LIN {X 0,Y 302.107,Z 503.378,A -85,B 0,C 180,E1 -16252.782,E2 -16252.782} C_VEL
LIN {X 0,Y 301.296,Z 506.672,A -85,B 0,C 180,E1 -16255.913,E2 -16255.913} C_VEL
LIN {X 0,Y 301.67,Z 508.867,A -85,B 0,C 180,E1 -16256.346,E2 -16256.346} C_VEL
LIN {X 0,Y 303.743,Z 513.97,A -85,B 0,C 180,E1 -16257.676,E2 -16257.676} C_VEL
LIN {X 0,Y 305.482,Z 519.047,A -85,B 0,C 180,E1 -16258.793,E2 -16258.793} C_VEL
LIN {X 0,Y 308.802,Z 531.713,A -85,B 0,C 180,E1 -16261.229,E2 -16261.229} C_VEL
LIN {X 0,Y 310.479,Z 540.82,A -85,B 0,C 180,E1 -16262.787,E2 -16262.787} C_VEL
LIN {X 0,Y 311.403,Z 551.592,A -85,B 0,C 180,E1 -16264.523,E2 -16264.523} C_VEL
LIN {X 0,Y 311.098,Z 562.085,A -85,B 0,C 180,E1 -16266.183,E2 -16266.183} C_VEL
LIN {X 0,Y 309.471,Z 571.424,A -85,B 0,C 180,E1 -16267.642,E2 -16267.642} C_VEL
LIN {X 0,Y 306.369,Z 582.24,A -85,B 0,C 180,E1 -16269.523,E2 -16269.523} C_VEL
LIN {X 0,Y 304.149,Z 589.898,A -85,B 0,C 180,E1 -16271.125,E2 -16271.125} C_VEL
LIN {X 0,Y 301.756,Z 598.006,A -85,B 0,C 180,E1 -16273.167,E2 -16273.167} C_VEL
LIN {X 0,Y 299.626,Z 606.028,A -85,B 0,C 180,E1 -16275.742,E2 -16275.742} C_VEL
LIN {X 0,Y 298.242,Z 611.012,A -85,B 0,C 180,E1 -16277.755,E2 -16277.755} C_VEL
LIN {X 0,Y 297.426,Z 614.951,A -85,B 0,C 180,E1 -16279.792,E2 -16279.792} C_VEL
LIN {X 0,Y 296.891,Z 617.952,A -85,B 0,C 180,E1 -16281.834,E2 -16281.834} C_VEL
LIN {X 0,Y 296.6,Z 620.554,A -85,B 0,C 180,E1 -16284.561,E2 -16284.561} C_VEL
LIN {X 0,Y 296.644,Z 621.226,A -85,B 0,C 180,E1 -16285.924,E2 -16285.924} C_VEL
LIN {X 0,Y 296.862,Z 621.354,A -85,B 0,C 180,E1 -16288.643,E2 -16288.643} C_VEL
LIN {X 0,Y 296.994,Z 620.811,A -85,B 0,C 180,E1 -16290,E2 -16290} C_VEL
LIN {X 0,Y 296.996,Z 619.807,A -85,B 0,C 180,E1 -16291.356,E2 -16291.356} C_VEL
LIN {X 0,Y 296.811,Z 618.326,A -85,B 0,C 180,E1 -16292.714,E2 -16292.714} C_VEL
LIN {X 0,Y 296.889,Z 615.286,A -85,B 0,C 180,E1 -16294.752,E2 -16294.752} C_VEL
LIN {X 0,Y 296.979,Z 611.114,A -85,B 0,C 180,E1 -16296.795,E2 -16296.795} C_VEL
LIN {X 0,Y 297.198,Z 604.706,A -85,B 0,C 180,E1 -16299.185,E2 -16299.185} C_VEL
LIN {X 0,Y 297.65,Z 597.649,A -85,B 0,C 180,E1 -16301.233,E2 -16301.233} C_VEL
LIN {X 0,Y 298.482,Z 588.932,A -85,B 0,C 180,E1 -16303.272,E2 -16303.272} C_VEL
LIN {X 0,Y 299.3,Z 580.046,A -85,B 0,C 180,E1 -16304.969,E2 -16304.969} C_VEL
LIN {X 0,Y 300.483,Z 569.203,A -85,B 0,C 180,E1 -16306.649,E2 -16306.649} C_VEL
LIN {X 0,Y 301.456,Z 558.568,A -85,B 0,C 180,E1 -16307.993,E2 -16307.993} C_VEL
LIN {X 0,Y 300.374,Z 546.843,A -85,B 0,C 180,E1 -16309.237,E2 -16309.237} C_VEL
LIN {X 0,Y 299.033,Z 533.574,A -85,B 0,C 180,E1 -16310.352,E2 -16310.352} C_VEL
LIN {X 0,Y 297.686,Z 520.117,A -85,B 0,C 180,E1 -16311.216,E2 -16311.216} C_VEL
LIN {X 0,Y 297.486,Z 517.081,A -85,B 0,C 180,E1 -16311.389,E2 -16311.389} C_VEL
LIN {X 0,Y 298.225,Z 509.911,A -85,B 0,C 180,E1 -16315.793,E2 -16315.793} C_VEL
LIN {X 0,Y 299.087,Z 503.762,A -85,B 0,C 180,E1 -16319.607,E2 -16319.607} C_VEL
LIN {X 0,Y 300.024,Z 497.747,A -85,B 0,C 180,E1 -16323.4,E2 -16323.4} C_VEL
LIN {X 0,Y 300.596,Z 494.041,A -85,B 0,C 180,E1 -16325.768,E2 -16325.768} C_VEL
LIN {X 0,Y 300.422,Z 490.212,A -85,B 0,C 180,E1 -16328.311,E2 -16328.311} C_VEL
LIN {X 0,Y 299.452,Z 484.838,A -85,B 0,C 180,E1 -16332.082,E2 -16332.082} C_VEL
LIN {X 0,Y 298.523,Z 479.301,A -85,B 0,C 180,E1 -16336.189,E2 -16336.189} C_VEL
LIN {X 0,Y 298.427,Z 479.312,A -85,B 0,C 180,E1 -16340.517,E2 -16340.517} C_VEL
LIN {X 0,Y 298.432,Z 479.308,A -85,B 0,C 180,E1 -16343.932,E2 -16343.932} C_VEL
LIN {X 0,Y 298.394,Z 479.313,A -85,B 0,C 180,E1 -16347.984,E2 -16347.984} C_VEL
LIN {X 0,Y 298.458,Z 479.304,A -85,B 0,C 180,E1 -16351.904,E2 -16351.904} C_VEL
LIN {X 0,Y 298.484,Z 479.304,A -85,B 0,C 180,E1 -16354.924,E2 -16354.924} C_VEL
LIN {X 0,Y 298.451,Z 479.305,A -85,B 0,C 180,E1 -16359.316,E2 -16359.316} C_VEL
LIN {X 0,Y 298.539,Z 479.296,A -85,B 0,C 180,E1 -16362.18,E2 -16362.18} C_VEL
LIN {X 0,Y 298.595,Z 479.29,A -85,B 0,C 180,E1 -16364.995,E2 -16364.995} C_VEL
LIN {X 0,Y 298.595,Z 479.288,A -85,B 0,C 180,E1 -16369.147,E2 -16369.147} C_VEL
LIN {X 0,Y 298.76,Z 479.268,A -85,B 0,C 180,E1 -16371.886,E2 -16371.886} C_VEL
LIN {X 0,Y 298.661,Z 479.284,A -85,B 0,C 180,E1 -16374.599,E2 -16374.599} C_VEL
LIN {X 0,Y 298.925,Z 479.25,A -85,B 0,C 180,E1 -16378.653,E2 -16378.653} C_VEL
LIN {X 0,Y 298.926,Z 479.247,A -85,B 0,C 180,E1 -16381.347,E2 -16381.347} C_VEL
LIN {X 0,Y 298.8,Z 479.264,A -85,B 0,C 180,E1 -16386.754,E2 -16386.754} C_VEL
LIN {X 0,Y 298.682,Z 479.277,A -85,B 0,C 180,E1 -16389.481,E2 -16389.481} C_VEL
LIN {X 0,Y 298.554,Z 479.293,A -85,B 0,C 180,E1 -16393.616,E2 -16393.616} C_VEL
LIN {X 0,Y 298.55,Z 479.298,A -85,B 0,C 180,E1 -16396.409,E2 -16396.409} C_VEL
LIN {X 0,Y 298.514,Z 479.298,A -85,B 0,C 180,E1 -16399.655,E2 -16399.655} C_VEL
LIN {X 0,Y 298.459,Z 479.304,A -85,B 0,C 180,E1 -16403.598,E2 -16403.598} C_VEL
LIN {X 0,Y 298.491,Z 479.304,A -85,B 0,C 180,E1 -16406.575,E2 -16406.575} C_VEL
LIN {X 0,Y 298.423,Z 479.31,A -85,B 0,C 180,E1 -16409.641,E2 -16409.641} C_VEL
LIN {X 0,Y 298.398,Z 479.313,A -85,B 0,C 180,E1 -16412.8,E2 -16412.8} C_VEL
LIN {X 0,Y 298.448,Z 479.307,A -85,B 0,C 180,E1 -16416.808,E2 -16416.808} C_VEL
LIN {X 0,Y 298.411,Z 479.311,A -85,B 0,C 180,E1 -16419.486,E2 -16419.486} C_VEL
LIN {X 0,Y 298.4,Z 479.312,A -85,B 0,C 180,E1 -16423.104,E2 -16423.104} C_VEL
LIN {X 0,Y 298.405,Z 479.312,A -85,B 0,C 180,E1 -16426.921,E2 -16426.921} C_VEL
LIN {X 0,Y 298.418,Z 479.309,A -85,B 0,C 180,E1 -16431.004,E2 -16431.004} C_VEL
LIN {X 0,Y 298.435,Z 479.311,A -85,B 0,C 180,E1 -16433.933,E2 -16433.933} C_VEL
LIN {X 0,Y 298.397,Z 479.316,A -85,B 0,C 180,E1 -16437.984,E2 -16437.984} C_VEL
LIN {X 0,Y 298.462,Z 479.307,A -85,B 0,C 180,E1 -16441.904,E2 -16441.904} C_VEL
LIN {X 0,Y 298.489,Z 479.301,A -85,B 0,C 180,E1 -16444.924,E2 -16444.924} C_VEL
LIN {X 0,Y 298.454,Z 479.305,A -85,B 0,C 180,E1 -16449.316,E2 -16449.316} C_VEL
LIN {X 0,Y 298.542,Z 479.299,A -85,B 0,C 180,E1 -16452.18,E2 -16452.18} C_VEL
LIN {X 0,Y 298.597,Z 479.287,A -85,B 0,C 180,E1 -16454.995,E2 -16454.995} C_VEL
LIN {X 0,Y 298.595,Z 479.288,A -85,B 0,C 180,E1 -16459.147,E2 -16459.147} C_VEL
LIN {X 0,Y 298.717,Z 479.276,A -85,B 0,C 180,E1 -16461.885,E2 -16461.885} C_VEL
LIN {X 0,Y 298.648,Z 479.281,A -85,B 0,C 180,E1 -16464.599,E2 -16464.599} C_VEL
LIN {X 0,Y 298.928,Z 479.247,A -85,B 0,C 180,E1 -16468.653,E2 -16468.653} C_VEL
LIN {X 0,Y 298.926,Z 479.247,A -85,B 0,C 180,E1 -16471.347,E2 -16471.347} C_VEL
LIN {X 0,Y 298.791,Z 479.263,A -85,B 0,C 180,E1 -16476.754,E2 -16476.754} C_VEL
LIN {X 0,Y 298.64,Z 479.284,A -85,B 0,C 180,E1 -16479.482,E2 -16479.482} C_VEL
LIN {X 0,Y 298.556,Z 479.294,A -85,B 0,C 180,E1 -16483.615,E2 -16483.615} C_VEL
LIN {X 0,Y 298.553,Z 479.294,A -85,B 0,C 180,E1 -16486.409,E2 -16486.409} C_VEL
LIN {X 0,Y 298.516,Z 479.301,A -85,B 0,C 180,E1 -16489.655,E2 -16489.655} C_VEL
LIN {X 0,Y 298.461,Z 479.307,A -85,B 0,C 180,E1 -16493.598,E2 -16493.598} C_VEL
LIN {X 0,Y 298.49,Z 479.301,A -85,B 0,C 180,E1 -16496.575,E2 -16496.575} C_VEL
LIN {X 0,Y 298.42,Z 479.313,A -85,B 0,C 180,E1 -16499.641,E2 -16499.641} C_VEL
LIN {X 0,Y 298.399,Z 479.312,A -85,B 0,C 180,E1 -16502.8,E2 -16502.8} C_VEL
LIN {X 0,Y 298.454,Z 479.305,A -85,B 0,C 180,E1 -16506.809,E2 -16506.809} C_VEL
LIN {X 0,Y 298.412,Z 479.313,A -85,B 0,C 180,E1 -16509.486,E2 -16509.486} C_VEL
LIN {X 0,Y 298.402,Z 479.312,A -85,B 0,C 180,E1 -16513.103,E2 -16513.103} C_VEL
LIN {X 0,Y 298.406,Z 479.311,A -85,B 0,C 180,E1 -16516.921,E2 -16516.921} C_VEL
LIN {X 0,Y 298.392,Z 479.313,A -85,B 0,C 180,E1 -16521.01,E2 -16521.01} C_VEL
LIN {X 0,Y 298.304,Z 479.327,A -85,B 0,C 180,E1 -16523.914,E2 -16523.914} C_VEL
LIN {X 0,Y 297.986,Z 479.364,A -85,B 0,C 180,E1 -16527.149,E2 -16527.149} C_VEL
LIN {X 0,Y 297.642,Z 479.407,A -85,B 0,C 180,E1 -16530.887,E2 -16530.887} C_VEL
LIN {X 0,Y 297.319,Z 479.451,A -85,B 0,C 180,E1 -16533.928,E2 -16533.928} C_VEL
LIN {X 0,Y 297.221,Z 479.745,A -85,B 0,C 180,E1 -16534.81,E2 -16534.81} C_VEL
LIN {X 0,Y 297.105,Z 483.567,A -85,B 0,C 180,E1 -16538.89,E2 -16538.89} C_VEL
LIN {X 0,Y 299.629,Z 496.768,A -85,B 0,C 180,E1 -16539.757,E2 -16539.757} C_VEL
LIN {X 0,Y 302.182,Z 509.983,A -85,B 0,C 180,E1 -16540.89,E2 -16540.89} C_VEL
LIN {X 0,Y 302.831,Z 515.047,A -85,B 0,C 180,E1 -16541.391,E2 -16541.391} C_VEL
LIN {X 0,Y 301.789,Z 527.176,A -85,B 0,C 180,E1 -16542.709,E2 -16542.709} C_VEL
LIN {X 0,Y 300.718,Z 538.429,A -85,B 0,C 180,E1 -16544.235,E2 -16544.235} C_VEL
LIN {X 0,Y 299.799,Z 547.646,A -85,B 0,C 180,E1 -16545.75,E2 -16545.75} C_VEL
LIN {X 0,Y 298.768,Z 557.725,A -85,B 0,C 180,E1 -16547.777,E2 -16547.777} C_VEL
LIN {X 0,Y 298,Z 565.938,A -85,B 0,C 180,E1 -16549.812,E2 -16549.812} C_VEL
LIN {X 0,Y 297.448,Z 572.604,A -85,B 0,C 180,E1 -16551.85,E2 -16551.85} C_VEL
LIN {X 0,Y 297.056,Z 578.093,A -85,B 0,C 180,E1 -16553.957,E2 -16553.957} C_VEL
LIN {X 0,Y 296.938,Z 582.134,A -85,B 0,C 180,E1 -16555.928,E2 -16555.928} C_VEL
LIN {X 0,Y 296.865,Z 583.076,A -85,B 0,C 180,E1 -16556.475,E2 -16556.475} C_VEL
LIN {X 0,Y 296.11,Z 584.795,A -85,B 0,C 180,E1 -16557.557,E2 -16557.557} C_VEL
LIN {X 0,Y 293.211,Z 587.005,A -85,B 0,C 180,E1 -16559.351,E2 -16559.351} C_VEL
LIN {X 0,Y 290.88,Z 588.266,A -85,B 0,C 180,E1 -16560.828,E2 -16560.828} C_VEL
LIN {X 0,Y 289.989,Z 588.981,A -85,B 0,C 180,E1 -16561.979,E2 -16561.979} C_VEL
LIN {X 0,Y 289.972,Z 589.117,A -85,B 0,C 180,E1 -16562.369,E2 -16562.369} C_VEL
LIN {X 0,Y 290.338,Z 589.507,A -85,B 0,C 180,E1 -16564.164,E2 -16564.164} C_VEL
LIN {X 0,Y 290.839,Z 588.823,A -85,B 0,C 180,E1 -16566.939,E2 -16566.939} C_VEL
LIN {X 0,Y 292.244,Z 586.468,A -85,B 0,C 180,E1 -16569.691,E2 -16569.691} C_VEL
LIN {X 0,Y 293.876,Z 582.596,A -85,B 0,C 180,E1 -16572.429,E2 -16572.429} C_VEL
LIN {X 0,Y 295.649,Z 578.513,A -85,B 0,C 180,E1 -16574.454,E2 -16574.454} C_VEL
LIN {X 0,Y 297.634,Z 573.361,A -85,B 0,C 180,E1 -16576.46,E2 -16576.46} C_VEL
LIN {X 0,Y 300.395,Z 565.915,A -85,B 0,C 180,E1 -16578.765,E2 -16578.765} C_VEL
LIN {X 0,Y 303.37,Z 557.96,A -85,B 0,C 180,E1 -16580.688,E2 -16580.688} C_VEL
LIN {X 0,Y 306.517,Z 548.367,A -85,B 0,C 180,E1 -16582.585,E2 -16582.585} C_VEL
LIN {X 0,Y 309.442,Z 538.773,A -85,B 0,C 180,E1 -16584.13,E2 -16584.13} C_VEL
LIN {X 0,Y 310.422,Z 534.633,A -85,B 0,C 180,E1 -16584.744,E2 -16584.744} C_VEL
LIN {X 0,Y 308.526,Z 525.506,A -85,B 0,C 180,E1 -16586.831,E2 -16586.831} C_VEL
LIN {X 0,Y 306.405,Z 519.377,A -85,B 0,C 180,E1 -16588.413,E2 -16588.413} C_VEL
LIN {X 0,Y 303.715,Z 513.027,A -85,B 0,C 180,E1 -16590.241,E2 -16590.241} C_VEL
LIN {X 0,Y 302.235,Z 509.907,A -85,B 0,C 180,E1 -16591.215,E2 -16591.215} C_VEL
LIN {X 0,Y 300.186,Z 506.257,A -85,B 0,C 180,E1 -16592.58,E2 -16592.58} C_VEL
LIN {X 0,Y 298.449,Z 503.948,A -85,B 0,C 180,E1 -16593.694,E2 -16593.694} C_VEL
LIN {X 0,Y 297.462,Z 501.682,A -85,B 0,C 180,E1 -16594.544,E2 -16594.544} C_VEL
LIN {X 0,Y 295.377,Z 499.782,A -85,B 0,C 180,E1 -16596.004,E2 -16596.004} C_VEL
LIN {X 0,Y 294.153,Z 496.998,A -85,B 0,C 180,E1 -16597.437,E2 -16597.437} C_VEL
LIN {X 0,Y 294.39,Z 497.575,A -85,B 0,C 180,E1 -16600.187,E2 -16600.187} C_VEL
LIN {X 0,Y 294.661,Z 498.846,A -85,B 0,C 180,E1 -16603.764,E2 -16603.764} C_VEL
LIN {X 0,Y 295.006,Z 500.89,A -85,B 0,C 180,E1 -16607.606,E2 -16607.606} C_VEL
LIN {X 0,Y 295.213,Z 502.538,A -85,B 0,C 180,E1 -16610,E2 -16610} C_VEL
LIN {X 0,Y 295.074,Z 505.124,A -85,B 0,C 180,E1 -16613.035,E2 -16613.035} C_VEL
LIN {X 0,Y 295.688,Z 508.225,A -85,B 0,C 180,E1 -16613.913,E2 -16613.913} C_VEL
LIN {X 0,Y 297.728,Z 512.868,A -85,B 0,C 180,E1 -16615.491,E2 -16615.491} C_VEL
LIN {X 0,Y 298.885,Z 516.803,A -85,B 0,C 180,E1 -16616.493,E2 -16616.493} C_VEL
LIN {X 0,Y 299.627,Z 518.634,A -85,B 0,C 180,E1 -16617.017,E2 -16617.017} C_VEL
LIN {X 0,Y 301.626,Z 526.286,A -85,B 0,C 180,E1 -16618.733,E2 -16618.733} C_VEL
LIN {X 0,Y 303.297,Z 533.136,A -85,B 0,C 180,E1 -16620.169,E2 -16620.169} C_VEL
LIN {X 0,Y 304.843,Z 542.716,A -85,B 0,C 180,E1 -16621.97,E2 -16621.97} C_VEL
LIN {X 0,Y 305.551,Z 553.087,A -85,B 0,C 180,E1 -16623.772,E2 -16623.772} C_VEL
LIN {X 0,Y 305.105,Z 563.405,A -85,B 0,C 180,E1 -16625.504,E2 -16625.504} C_VEL
LIN {X 0,Y 303.053,Z 573.235,A -85,B 0,C 180,E1 -16627.142,E2 -16627.142} C_VEL
LIN {X 0,Y 299.851,Z 583.62,A -85,B 0,C 180,E1 -16629.057,E2 -16629.057} C_VEL
LIN {X 0,Y 297.012,Z 592.414,A -85,B 0,C 180,E1 -16631.057,E2 -16631.057} C_VEL
LIN {X 0,Y 294.771,Z 599.512,A -85,B 0,C 180,E1 -16633.018,E2 -16633.018} C_VEL
LIN {X 0,Y 292.767,Z 606.445,A -85,B 0,C 180,E1 -16635.4,E2 -16635.4} C_VEL
LIN {X 0,Y 291.287,Z 611.213,A -85,B 0,C 180,E1 -16637.458,E2 -16637.458} C_VEL
LIN {X 0,Y 290.195,Z 616.022,A -85,B 0,C 180,E1 -16640.239,E2 -16640.239} C_VEL
LIN {X 0,Y 289.605,Z 619.229,A -85,B 0,C 180,E1 -16643.031,E2 -16643.031} C_VEL
LIN {X 0,Y 289.536,Z 620.209,A -85,B 0,C 180,E1 -16644.428,E2 -16644.428} C_VEL
LIN {X 0,Y 289.555,Z 620.796,A -85,B 0,C 180,E1 -16645.824,E2 -16645.824} C_VEL
LIN {X 0,Y 289.773,Z 620.785,A -85,B 0,C 180,E1 -16648.61,E2 -16648.61} C_VEL
LIN {X 0,Y 289.94,Z 620.14,A -85,B 0,C 180,E1 -16650,E2 -16650} C_VEL
LIN {X 0,Y 289.938,Z 619.046,A -85,B 0,C 180,E1 -16651.389,E2 -16651.389} C_VEL
LIN {X 0,Y 289.741,Z 617.499,A -85,B 0,C 180,E1 -16652.78,E2 -16652.78} C_VEL
LIN {X 0,Y 289.839,Z 614.321,A -85,B 0,C 180,E1 -16654.868,E2 -16654.868} C_VEL
LIN {X 0,Y 289.926,Z 610.008,A -85,B 0,C 180,E1 -16656.961,E2 -16656.961} C_VEL
LIN {X 0,Y 290.174,Z 603.387,A -85,B 0,C 180,E1 -16659.409,E2 -16659.409} C_VEL
LIN {X 0,Y 290.668,Z 596.139,A -85,B 0,C 180,E1 -16661.506,E2 -16661.506} C_VEL
LIN {X 0,Y 291.538,Z 587.211,A -85,B 0,C 180,E1 -16663.594,E2 -16663.594} C_VEL
LIN {X 0,Y 292.568,Z 576.541,A -85,B 0,C 180,E1 -16665.583,E2 -16665.583} C_VEL
LIN {X 0,Y 293.789,Z 565.673,A -85,B 0,C 180,E1 -16667.219,E2 -16667.219} C_VEL
LIN {X 0,Y 294.292,Z 557.319,A -85,B 0,C 180,E1 -16668.266,E2 -16668.266} C_VEL
LIN {X 0,Y 293.043,Z 544.534,A -85,B 0,C 180,E1 -16669.619,E2 -16669.619} C_VEL
LIN {X 0,Y 291.658,Z 530.634,A -85,B 0,C 180,E1 -16670.777,E2 -16670.777} C_VEL
LIN {X 0,Y 290.419,Z 516.721,A -85,B 0,C 180,E1 -16671.656,E2 -16671.656} C_VEL
LIN {X 0,Y 291.116,Z 510.248,A -85,B 0,C 180,E1 -16675.756,E2 -16675.756} C_VEL
LIN {X 0,Y 292.082,Z 503.639,A -85,B 0,C 180,E1 -16679.977,E2 -16679.977} C_VEL
LIN {X 0,Y 293.164,Z 496.988,A -85,B 0,C 180,E1 -16684.289,E2 -16684.289} C_VEL
LIN {X 0,Y 293.549,Z 493.273,A -85,B 0,C 180,E1 -16686.765,E2 -16686.765} C_VEL
LIN {X 0,Y 292.981,Z 488.85,A -85,B 0,C 180,E1 -16689.86,E2 -16689.86} C_VEL
LIN {X 0,Y 292.002,Z 483.47,A -85,B 0,C 180,E1 -16693.776,E2 -16693.776} C_VEL
LIN {X 0,Y 291.486,Z 480.178,A -85,B 0,C 180,E1 -16696.33,E2 -16696.33} C_VEL
LIN {X 0,Y 291.403,Z 480.187,A -85,B 0,C 180,E1 -16700.513,E2 -16700.513} C_VEL
LIN {X 0,Y 291.428,Z 480.183,A -85,B 0,C 180,E1 -16702.923,E2 -16702.923} C_VEL
LIN {X 0,Y 291.345,Z 480.193,A -85,B 0,C 180,E1 -16706.302,E2 -16706.302} C_VEL
LIN {X 0,Y 291.384,Z 480.188,A -85,B 0,C 180,E1 -16710.261,E2 -16710.261} C_VEL
LIN {X 0,Y 291.413,Z 480.184,A -85,B 0,C 180,E1 -16714.272,E2 -16714.272} C_VEL
LIN {X 0,Y 291.383,Z 480.187,A -85,B 0,C 180,E1 -16717.3,E2 -16717.3} C_VEL
LIN {X 0,Y 291.459,Z 480.178,A -85,B 0,C 180,E1 -16720.27,E2 -16720.27} C_VEL
LIN {X 0,Y 291.556,Z 480.17,A -85,B 0,C 180,E1 -16724.624,E2 -16724.624} C_VEL
LIN {X 0,Y 291.538,Z 480.168,A -85,B 0,C 180,E1 -16728.881,E2 -16728.881} C_VEL
LIN {X 0,Y 291.71,Z 480.145,A -85,B 0,C 180,E1 -16731.689,E2 -16731.689} C_VEL
LIN {X 0,Y 291.632,Z 480.16,A -85,B 0,C 180,E1 -16734.469,E2 -16734.469} C_VEL
LIN {X 0,Y 291.891,Z 480.127,A -85,B 0,C 180,E1 -16738.621,E2 -16738.621} C_VEL
LIN {X 0,Y 291.892,Z 480.123,A -85,B 0,C 180,E1 -16741.38,E2 -16741.38} C_VEL
LIN {X 0,Y 291.748,Z 480.142,A -85,B 0,C 180,E1 -16746.918,E2 -16746.918} C_VEL
LIN {X 0,Y 291.631,Z 480.156,A -85,B 0,C 180,E1 -16749.712,E2 -16749.712} C_VEL
LIN {X 0,Y 291.524,Z 480.17,A -85,B 0,C 180,E1 -16753.951,E2 -16753.951} C_VEL
LIN {X 0,Y 291.489,Z 480.175,A -85,B 0,C 180,E1 -16756.818,E2 -16756.818} C_VEL
LIN {X 0,Y 291.452,Z 480.179,A -85,B 0,C 180,E1 -16759.875,E2 -16759.875} C_VEL
LIN {X 0,Y 291.402,Z 480.187,A -85,B 0,C 180,E1 -16764.205,E2 -16764.205} C_VEL
LIN {X 0,Y 291.424,Z 480.181,A -85,B 0,C 180,E1 -16767.272,E2 -16767.272} C_VEL
LIN {X 0,Y 291.339,Z 480.195,A -85,B 0,C 180,E1 -16770.437,E2 -16770.437} C_VEL
LIN {X 0,Y 291.347,Z 480.19,A -85,B 0,C 180,E1 -16773.699,E2 -16773.699} C_VEL
LIN {X 0,Y 291.383,Z 480.186,A -85,B 0,C 180,E1 -16777.256,E2 -16777.256} C_VEL
LIN {X 0,Y 291.336,Z 480.193,A -85,B 0,C 180,E1 -16780.643,E2 -16780.643} C_VEL
LIN {X 0,Y 291.292,Z 480.201,A -85,B 0,C 180,E1 -16784.402,E2 -16784.402} C_VEL
LIN {X 0,Y 291.329,Z 480.196,A -85,B 0,C 180,E1 -16788.405,E2 -16788.405} C_VEL
LIN {X 0,Y 291.367,Z 480.187,A -85,B 0,C 180,E1 -16791.161,E2 -16791.161} C_VEL
LIN {X 0,Y 291.388,Z 480.187,A -85,B 0,C 180,E1 -16794.63,E2 -16794.63} C_VEL
LIN {X 0,Y 291.374,Z 480.19,A -85,B 0,C 180,E1 -16797.951,E2 -16797.951} C_VEL
LIN {X 0,Y 291.38,Z 480.186,A -85,B 0,C 180,E1 -16801.158,E2 -16801.158} C_VEL
LIN {X 0,Y 291.418,Z 480.186,A -85,B 0,C 180,E1 -16804.272,E2 -16804.272} C_VEL
LIN {X 0,Y 291.385,Z 480.185,A -85,B 0,C 180,E1 -16807.3,E2 -16807.3} C_VEL
LIN {X 0,Y 291.462,Z 480.18,A -85,B 0,C 180,E1 -16810.271,E2 -16810.271} C_VEL
LIN {X 0,Y 291.559,Z 480.165,A -85,B 0,C 180,E1 -16814.624,E2 -16814.624} C_VEL
LIN {X 0,Y 291.539,Z 480.167,A -85,B 0,C 180,E1 -16818.881,E2 -16818.881} C_VEL
LIN {X 0,Y 291.668,Z 480.153,A -85,B 0,C 180,E1 -16821.687,E2 -16821.687} C_VEL
LIN {X 0,Y 291.617,Z 480.158,A -85,B 0,C 180,E1 -16824.468,E2 -16824.468} C_VEL
LIN {X 0,Y 291.894,Z 480.123,A -85,B 0,C 180,E1 -16828.62,E2 -16828.62} C_VEL
LIN {X 0,Y 291.893,Z 480.123,A -85,B 0,C 180,E1 -16831.38,E2 -16831.38} C_VEL
LIN {X 0,Y 291.739,Z 480.142,A -85,B 0,C 180,E1 -16836.918,E2 -16836.918} C_VEL
LIN {X 0,Y 291.579,Z 480.165,A -85,B 0,C 180,E1 -16839.714,E2 -16839.714} C_VEL
LIN {X 0,Y 291.526,Z 480.173,A -85,B 0,C 180,E1 -16843.95,E2 -16843.95} C_VEL
LIN {X 0,Y 291.491,Z 480.173,A -85,B 0,C 180,E1 -16846.818,E2 -16846.818} C_VEL
LIN {X 0,Y 291.454,Z 480.182,A -85,B 0,C 180,E1 -16849.875,E2 -16849.875} C_VEL
LIN {X 0,Y 291.404,Z 480.186,A -85,B 0,C 180,E1 -16854.205,E2 -16854.205} C_VEL
LIN {X 0,Y 291.423,Z 480.182,A -85,B 0,C 180,E1 -16857.272,E2 -16857.272} C_VEL
LIN {X 0,Y 291.338,Z 480.191,A -85,B 0,C 180,E1 -16860.437,E2 -16860.437} C_VEL
LIN {X 0,Y 291.348,Z 480.194,A -85,B 0,C 180,E1 -16863.698,E2 -16863.698} C_VEL
LIN {X 0,Y 291.388,Z 480.187,A -85,B 0,C 180,E1 -16867.256,E2 -16867.256} C_VEL
LIN {X 0,Y 291.337,Z 480.191,A -85,B 0,C 180,E1 -16870.642,E2 -16870.642} C_VEL
LIN {X 0,Y 291.293,Z 480.198,A -85,B 0,C 180,E1 -16874.402,E2 -16874.402} C_VEL
LIN {X 0,Y 291.329,Z 480.192,A -85,B 0,C 180,E1 -16878.404,E2 -16878.404} C_VEL
LIN {X 0,Y 291.338,Z 480.193,A -85,B 0,C 180,E1 -16881.155,E2 -16881.155} C_VEL
LIN {X 0,Y 291.33,Z 480.193,A -85,B 0,C 180,E1 -16882.907,E2 -16882.907} C_VEL
LIN {X 0,Y 291.028,Z 480.23,A -85,B 0,C 180,E1 -16886.26,E2 -16886.26} C_VEL
LIN {X 0,Y 290.709,Z 480.273,A -85,B 0,C 180,E1 -16889.49,E2 -16889.49} C_VEL
LIN {X 0,Y 290.366,Z 480.319,A -85,B 0,C 180,E1 -16892.621,E2 -16892.621} C_VEL
LIN {X 0,Y 290.238,Z 480.333,A -85,B 0,C 180,E1 -16894.159,E2 -16894.159} C_VEL
LIN {X 0,Y 290.085,Z 481.171,A -85,B 0,C 180,E1 -16895.678,E2 -16895.678} C_VEL
LIN {X 0,Y 290.038,Z 483.915,A -85,B 0,C 180,E1 -16898.64,E2 -16898.64} C_VEL
LIN {X 0,Y 292.535,Z 497.318,A -85,B 0,C 180,E1 -16899.547,E2 -16899.547} C_VEL
LIN {X 0,Y 295.269,Z 511.479,A -85,B 0,C 180,E1 -16900.806,E2 -16900.806} C_VEL
LIN {X 0,Y 295.769,Z 516.21,A -85,B 0,C 180,E1 -16901.289,E2 -16901.289} C_VEL
LIN {X 0,Y 294.616,Z 528.976,A -85,B 0,C 180,E1 -16902.748,E2 -16902.748} C_VEL
LIN {X 0,Y 293.562,Z 539.263,A -85,B 0,C 180,E1 -16904.197,E2 -16904.197} C_VEL
LIN {X 0,Y 292.662,Z 548.424,A -85,B 0,C 180,E1 -16905.75,E2 -16905.75} C_VEL
LIN {X 0,Y 291.654,Z 558.437,A -85,B 0,C 180,E1 -16907.828,E2 -16907.828} C_VEL
LIN {X 0,Y 290.874,Z 566.617,A -85,B 0,C 180,E1 -16909.911,E2 -16909.911} C_VEL
LIN {X 0,Y 290.393,Z 572.217,A -85,B 0,C 180,E1 -16911.65,E2 -16911.65} C_VEL
LIN {X 0,Y 289.95,Z 578.397,A -85,B 0,C 180,E1 -16914.03,E2 -16914.03} C_VEL
LIN {X 0,Y 289.789,Z 583.133,A -85,B 0,C 180,E1 -16916.452,E2 -16916.452} C_VEL
LIN {X 0,Y 289.673,Z 586.207,A -85,B 0,C 180,E1 -16918.61,E2 -16918.61} C_VEL
LIN {X 0,Y 289.71,Z 587.658,A -85,B 0,C 180,E1 -16920,E2 -16920} C_VEL
LIN {X 0,Y 289.972,Z 589.117,A -85,B 0,C 180,E1 -16922.369,E2 -16922.369} C_VEL
LIN {X 0,Y 289.5,Z 589.557,A -85,B 0,C 180,E1 -16923.53,E2 -16923.53} C_VEL
LIN {X 0,Y 286.985,Z 589.879,A -85,B 0,C 180,E1 -16925.438,E2 -16925.438} C_VEL
LIN {X 0,Y 284.676,Z 589.426,A -85,B 0,C 180,E1 -16927.374,E2 -16927.374} C_VEL
LIN {X 0,Y 284.537,Z 588.648,A -85,B 0,C 180,E1 -16928.554,E2 -16928.554} C_VEL
LIN {X 0,Y 285.319,Z 587.426,A -85,B 0,C 180,E1 -16929.929,E2 -16929.929} C_VEL
LIN {X 0,Y 287.054,Z 583.777,A -85,B 0,C 180,E1 -16932.729,E2 -16932.729} C_VEL
LIN {X 0,Y 288.927,Z 579.89,A -85,B 0,C 180,E1 -16934.798,E2 -16934.798} C_VEL
LIN {X 0,Y 291.043,Z 575.039,A -85,B 0,C 180,E1 -16936.844,E2 -16936.844} C_VEL
LIN {X 0,Y 293.932,Z 567.916,A -85,B 0,C 180,E1 -16939.194,E2 -16939.194} C_VEL
LIN {X 0,Y 297.604,Z 558.946,A -85,B 0,C 180,E1 -16941.471,E2 -16941.471} C_VEL
LIN {X 0,Y 300.924,Z 549.532,A -85,B 0,C 180,E1 -16943.393,E2 -16943.393} C_VEL
LIN {X 0,Y 304.704,Z 538.057,A -85,B 0,C 180,E1 -16945.266,E2 -16945.266} C_VEL
LIN {X 0,Y 303.91,Z 532.312,A -85,B 0,C 180,E1 -16946.62,E2 -16946.62} C_VEL
LIN {X 0,Y 302.341,Z 525.971,A -85,B 0,C 180,E1 -16948.288,E2 -16948.288} C_VEL
LIN {X 0,Y 299.317,Z 518.148,A -85,B 0,C 180,E1 -16950.686,E2 -16950.686} C_VEL
LIN {X 0,Y 296.222,Z 511.76,A -85,B 0,C 180,E1 -16953.071,E2 -16953.071} C_VEL
LIN {X 0,Y 293.909,Z 507.595,A -85,B 0,C 180,E1 -16955.022,E2 -16955.022} C_VEL
LIN {X 0,Y 292.51,Z 506.228,A -85,B 0,C 180,E1 -16956.139,E2 -16956.139} C_VEL
LIN {X 0,Y 291.532,Z 504.176,A -85,B 0,C 180,E1 -16957.294,E2 -16957.294} C_VEL
LIN {X 0,Y 289.809,Z 502.849,A -85,B 0,C 180,E1 -16959.103,E2 -16959.103} C_VEL
LIN {X 0,Y 288.536,Z 501.8,A -85,B 0,C 180,E1 -16961.121,E2 -16961.121} C_VEL
LIN {X 0,Y 287.962,Z 501.127,A -85,B 0,C 180,E1 -16963.107,E2 -16963.107} C_VEL
LIN {X 0,Y 287.906,Z 501.297,A -85,B 0,C 180,E1 -16965.065,E2 -16965.065} C_VEL
LIN {X 0,Y 288.19,Z 502.755,A -85,B 0,C 180,E1 -16967.021,E2 -16967.021} C_VEL
LIN {X 0,Y 288.898,Z 505.202,A -85,B 0,C 180,E1 -16968.95,E2 -16968.95} C_VEL
LIN {X 0,Y 291.868,Z 511.353,A -85,B 0,C 180,E1 -16972.619,E2 -16972.619} C_VEL
LIN {X 0,Y 292.809,Z 515.227,A -85,B 0,C 180,E1 -16973.863,E2 -16973.863} C_VEL
LIN {X 0,Y 294.015,Z 518.522,A -85,B 0,C 180,E1 -16974.992,E2 -16974.992} C_VEL
LIN {X 0,Y 295.856,Z 525.468,A -85,B 0,C 180,E1 -16976.882,E2 -16976.882} C_VEL
LIN {X 0,Y 297.626,Z 533.108,A -85,B 0,C 180,E1 -16978.701,E2 -16978.701} C_VEL
LIN {X 0,Y 299.177,Z 543.06,A -85,B 0,C 180,E1 -16980.781,E2 -16980.781} C_VEL
LIN {X 0,Y 299.837,Z 554.586,A -85,B 0,C 180,E1 -16982.961,E2 -16982.961} C_VEL
LIN {X 0,Y 299.205,Z 564.325,A -85,B 0,C 180,E1 -16984.719,E2 -16984.719} C_VEL
LIN {X 0,Y 297.302,Z 573.35,A -85,B 0,C 180,E1 -16986.305,E2 -16986.305} C_VEL
LIN {X 0,Y 293.877,Z 583.445,A -85,B 0,C 180,E1 -16988.242,E2 -16988.242} C_VEL
LIN {X 0,Y 290.895,Z 591.992,A -85,B 0,C 180,E1 -16990.23,E2 -16990.23} C_VEL
LIN {X 0,Y 288.374,Z 599.15,A -85,B 0,C 180,E1 -16992.263,E2 -16992.263} C_VEL
LIN {X 0,Y 286.477,Z 605.092,A -85,B 0,C 180,E1 -16994.344,E2 -16994.344} C_VEL
LIN {X 0,Y 284.799,Z 610.003,A -85,B 0,C 180,E1 -16996.442,E2 -16996.442} C_VEL
LIN {X 0,Y 283.704,Z 613.893,A -85,B 0,C 180,E1 -16998.569,E2 -16998.569} C_VEL
LIN {X 0,Y 282.795,Z 617.688,A -85,B 0,C 180,E1 -17001.424,E2 -17001.424} C_VEL
LIN {X 0,Y 282.482,Z 619.86,A -85,B 0,C 180,E1 -17004.288,E2 -17004.288} C_VEL
LIN {X 0,Y 282.471,Z 620.372,A -85,B 0,C 180,E1 -17005.719,E2 -17005.719} C_VEL
LIN {X 0,Y 282.5,Z 620.485,A -85,B 0,C 180,E1 -17007.148,E2 -17007.148} C_VEL
LIN {X 0,Y 282.704,Z 620.163,A -85,B 0,C 180,E1 -17008.575,E2 -17008.575} C_VEL
LIN {X 0,Y 282.885,Z 619.425,A -85,B 0,C 180,E1 -17010,E2 -17010} C_VEL
LIN {X 0,Y 282.88,Z 618.256,A -85,B 0,C 180,E1 -17011.423,E2 -17011.423} C_VEL
LIN {X 0,Y 282.686,Z 615.617,A -85,B 0,C 180,E1 -17013.563,E2 -17013.563} C_VEL
LIN {X 0,Y 282.848,Z 611.944,A -85,B 0,C 180,E1 -17015.704,E2 -17015.704} C_VEL
LIN {X 0,Y 282.913,Z 607.073,A -85,B 0,C 180,E1 -17017.853,E2 -17017.853} C_VEL
LIN {X 0,Y 283.213,Z 600.888,A -85,B 0,C 180,E1 -17020.003,E2 -17020.003} C_VEL
LIN {X 0,Y 283.842,Z 593.155,A -85,B 0,C 180,E1 -17022.149,E2 -17022.149} C_VEL
LIN {X 0,Y 284.759,Z 583.615,A -85,B 0,C 180,E1 -17024.288,E2 -17024.288} C_VEL
LIN {X 0,Y 285.852,Z 573.322,A -85,B 0,C 180,E1 -17026.144,E2 -17026.144} C_VEL
LIN {X 0,Y 287.085,Z 561.826,A -85,B 0,C 180,E1 -17027.819,E2 -17027.819} C_VEL
LIN {X 0,Y 287.174,Z 557.461,A -85,B 0,C 180,E1 -17028.366,E2 -17028.366} C_VEL
LIN {X 0,Y 285.961,Z 544.897,A -85,B 0,C 180,E1 -17029.751,E2 -17029.751} C_VEL
LIN {X 0,Y 284.642,Z 531.463,A -85,B 0,C 180,E1 -17030.922,E2 -17030.922} C_VEL
LIN {X 0,Y 283.377,Z 517.261,A -85,B 0,C 180,E1 -17031.84,E2 -17031.84} C_VEL
LIN {X 0,Y 283.353,Z 516.352,A -85,B 0,C 180,E1 -17031.937,E2 -17031.937} C_VEL
LIN {X 0,Y 284.156,Z 509.464,A -85,B 0,C 180,E1 -17036.436,E2 -17036.436} C_VEL
LIN {X 0,Y 285.068,Z 503.51,A -85,B 0,C 180,E1 -17040.358,E2 -17040.358} C_VEL
LIN {X 0,Y 286.116,Z 497.464,A -85,B 0,C 180,E1 -17044.399,E2 -17044.399} C_VEL
LIN {X 0,Y 286.486,Z 493.738,A -85,B 0,C 180,E1 -17046.943,E2 -17046.943} C_VEL
LIN {X 0,Y 285.974,Z 489.858,A -85,B 0,C 180,E1 -17049.715,E2 -17049.715} C_VEL
LIN {X 0,Y 284.991,Z 484.594,A -85,B 0,C 180,E1 -17053.669,E2 -17053.669} C_VEL
LIN {X 0,Y 284.433,Z 481.057,A -85,B 0,C 180,E1 -17056.447,E2 -17056.447} C_VEL
LIN {X 0,Y 284.352,Z 481.062,A -85,B 0,C 180,E1 -17060.013,E2 -17060.013} C_VEL
LIN {X 0,Y 284.352,Z 481.061,A -85,B 0,C 180,E1 -17063.617,E2 -17063.617} C_VEL
LIN {X 0,Y 284.308,Z 481.069,A -85,B 0,C 180,E1 -17067.19,E2 -17067.19} C_VEL
LIN {X 0,Y 284.356,Z 481.064,A -85,B 0,C 180,E1 -17070.376,E2 -17070.376} C_VEL
LIN {X 0,Y 284.375,Z 481.059,A -85,B 0,C 180,E1 -17073.586,E2 -17073.586} C_VEL
LIN {X 0,Y 284.368,Z 481.064,A -85,B 0,C 180,E1 -17076.707,E2 -17076.707} C_VEL
LIN {X 0,Y 284.404,Z 481.055,A -85,B 0,C 180,E1 -17081.262,E2 -17081.262} C_VEL
LIN {X 0,Y 284.493,Z 481.049,A -85,B 0,C 180,E1 -17084.459,E2 -17084.459} C_VEL
LIN {X 0,Y 284.49,Z 481.048,A -85,B 0,C 180,E1 -17088.602,E2 -17088.602} C_VEL
LIN {X 0,Y 284.66,Z 481.023,A -85,B 0,C 180,E1 -17091.481,E2 -17091.481} C_VEL
LIN {X 0,Y 284.603,Z 481.034,A -85,B 0,C 180,E1 -17094.332,E2 -17094.332} C_VEL
LIN {X 0,Y 284.857,Z 481.003,A -85,B 0,C 180,E1 -17098.586,E2 -17098.586} C_VEL
LIN {X 0,Y 284.858,Z 480.999,A -85,B 0,C 180,E1 -17101.414,E2 -17101.414} C_VEL
LIN {X 0,Y 284.7,Z 481.018,A -85,B 0,C 180,E1 -17107.09,E2 -17107.09} C_VEL
LIN {X 0,Y 284.568,Z 481.036,A -85,B 0,C 180,E1 -17109.956,E2 -17109.956} C_VEL
LIN {X 0,Y 284.483,Z 481.049,A -85,B 0,C 180,E1 -17114.303,E2 -17114.303} C_VEL
LIN {X 0,Y 284.427,Z 481.052,A -85,B 0,C 180,E1 -17117.249,E2 -17117.249} C_VEL
LIN {X 0,Y 284.38,Z 481.062,A -85,B 0,C 180,E1 -17120.242,E2 -17120.242} C_VEL
LIN {X 0,Y 284.371,Z 481.06,A -85,B 0,C 180,E1 -17123.876,E2 -17123.876} C_VEL
LIN {X 0,Y 284.399,Z 481.056,A -85,B 0,C 180,E1 -17127.174,E2 -17127.174} C_VEL
LIN {X 0,Y 284.298,Z 481.068,A -85,B 0,C 180,E1 -17131.274,E2 -17131.274} C_VEL
LIN {X 0,Y 284.343,Z 481.063,A -85,B 0,C 180,E1 -17135.348,E2 -17135.348} C_VEL
LIN {X 0,Y 284.321,Z 481.07,A -85,B 0,C 180,E1 -17138.168,E2 -17138.168} C_VEL
LIN {X 0,Y 284.271,Z 481.075,A -85,B 0,C 180,E1 -17142.125,E2 -17142.125} C_VEL
LIN {X 0,Y 284.258,Z 481.079,A -85,B 0,C 180,E1 -17146.19,E2 -17146.19} C_VEL
LIN {X 0,Y 284.309,Z 481.07,A -85,B 0,C 180,E1 -17150.024,E2 -17150.024} C_VEL
LIN {X 0,Y 284.353,Z 481.063,A -85,B 0,C 180,E1 -17153.617,E2 -17153.617} C_VEL
LIN {X 0,Y 284.31,Z 481.067,A -85,B 0,C 180,E1 -17157.19,E2 -17157.19} C_VEL
LIN {X 0,Y 284.358,Z 481.064,A -85,B 0,C 180,E1 -17160.376,E2 -17160.376} C_VEL
LIN {X 0,Y 284.379,Z 481.06,A -85,B 0,C 180,E1 -17163.587,E2 -17163.587} C_VEL
LIN {X 0,Y 284.37,Z 481.06,A -85,B 0,C 180,E1 -17166.707,E2 -17166.707} C_VEL
LIN {X 0,Y 284.407,Z 481.055,A -85,B 0,C 180,E1 -17171.262,E2 -17171.262} C_VEL
LIN {X 0,Y 284.496,Z 481.046,A -85,B 0,C 180,E1 -17174.459,E2 -17174.459} C_VEL
LIN {X 0,Y 284.491,Z 481.046,A -85,B 0,C 180,E1 -17178.602,E2 -17178.602} C_VEL
LIN {X 0,Y 284.623,Z 481.029,A -85,B 0,C 180,E1 -17181.48,E2 -17181.48} C_VEL
LIN {X 0,Y 284.586,Z 481.034,A -85,B 0,C 180,E1 -17184.331,E2 -17184.331} C_VEL
LIN {X 0,Y 284.86,Z 481,A -85,B 0,C 180,E1 -17188.586,E2 -17188.586} C_VEL
LIN {X 0,Y 284.859,Z 481,A -85,B 0,C 180,E1 -17191.414,E2 -17191.414} C_VEL
LIN {X 0,Y 284.69,Z 481.02,A -85,B 0,C 180,E1 -17197.09,E2 -17197.09} C_VEL
LIN {X 0,Y 284.523,Z 481.046,A -85,B 0,C 180,E1 -17199.957,E2 -17199.957} C_VEL
LIN {X 0,Y 284.486,Z 481.047,A -85,B 0,C 180,E1 -17204.303,E2 -17204.303} C_VEL
LIN {X 0,Y 284.43,Z 481.053,A -85,B 0,C 180,E1 -17207.248,E2 -17207.248} C_VEL
LIN {X 0,Y 284.382,Z 481.06,A -85,B 0,C 180,E1 -17210.242,E2 -17210.242} C_VEL
LIN {X 0,Y 284.373,Z 481.064,A -85,B 0,C 180,E1 -17213.876,E2 -17213.876} C_VEL
LIN {X 0,Y 284.399,Z 481.057,A -85,B 0,C 180,E1 -17217.173,E2 -17217.173} C_VEL
LIN {X 0,Y 284.298,Z 481.068,A -85,B 0,C 180,E1 -17221.274,E2 -17221.274} C_VEL
LIN {X 0,Y 284.345,Z 481.065,A -85,B 0,C 180,E1 -17225.348,E2 -17225.348} C_VEL
LIN {X 0,Y 284.323,Z 481.067,A -85,B 0,C 180,E1 -17228.168,E2 -17228.168} C_VEL
LIN {X 0,Y 284.272,Z 481.074,A -85,B 0,C 180,E1 -17232.124,E2 -17232.124} C_VEL
LIN {X 0,Y 284.258,Z 481.075,A -85,B 0,C 180,E1 -17236.189,E2 -17236.189} C_VEL
LIN {X 0,Y 284.309,Z 481.07,A -85,B 0,C 180,E1 -17240.024,E2 -17240.024} C_VEL
LIN {X 0,Y 284.21,Z 481.084,A -85,B 0,C 180,E1 -17243.595,E2 -17243.595} C_VEL
LIN {X 0,Y 283.904,Z 481.119,A -85,B 0,C 180,E1 -17247.317,E2 -17247.317} C_VEL
LIN {X 0,Y 283.61,Z 481.155,A -85,B 0,C 180,E1 -17250.29,E2 -17250.29} C_VEL
LIN {X 0,Y 283.257,Z 481.203,A -85,B 0,C 180,E1 -17253.474,E2 -17253.474} C_VEL
LIN {X 0,Y 283.053,Z 481.258,A -85,B 0,C 180,E1 -17255.033,E2 -17255.033} C_VEL
LIN {X 0,Y 282.976,Z 484.311,A -85,B 0,C 180,E1 -17258.38,E2 -17258.38} C_VEL
LIN {X 0,Y 285.46,Z 497.755,A -85,B 0,C 180,E1 -17259.319,E2 -17259.319} C_VEL
LIN {X 0,Y 288.07,Z 511.624,A -85,B 0,C 180,E1 -17260.585,E2 -17260.585} C_VEL
LIN {X 0,Y 288.753,Z 515.527,A -85,B 0,C 180,E1 -17261.002,E2 -17261.002} C_VEL
LIN {X 0,Y 287.666,Z 527.76,A -85,B 0,C 180,E1 -17262.394,E2 -17262.394} C_VEL
LIN {X 0,Y 286.559,Z 538.968,A -85,B 0,C 180,E1 -17263.983,E2 -17263.983} C_VEL
LIN {X 0,Y 285.528,Z 549.19,A -85,B 0,C 180,E1 -17265.75,E2 -17265.75} C_VEL
LIN {X 0,Y 284.52,Z 559.114,A -85,B 0,C 180,E1 -17267.88,E2 -17267.88} C_VEL
LIN {X 0,Y 283.725,Z 567.213,A -85,B 0,C 180,E1 -17270.015,E2 -17270.015} C_VEL
LIN {X 0,Y 283.224,Z 573.772,A -85,B 0,C 180,E1 -17272.156,E2 -17272.156} C_VEL
LIN {X 0,Y 282.847,Z 579.047,A -85,B 0,C 180,E1 -17274.296,E2 -17274.296} C_VEL
LIN {X 0,Y 282.716,Z 583.198,A -85,B 0,C 180,E1 -17276.437,E2 -17276.437} C_VEL
LIN {X 0,Y 282.586,Z 586.318,A -85,B 0,C 180,E1 -17278.575,E2 -17278.575} C_VEL
LIN {X 0,Y 282.752,Z 588.971,A -85,B 0,C 180,E1 -17281.424,E2 -17281.424} C_VEL
LIN {X 0,Y 282.971,Z 589.71,A -85,B 0,C 180,E1 -17282.847,E2 -17282.847} C_VEL
LIN {X 0,Y 283.267,Z 590.016,A -85,B 0,C 180,E1 -17284.268,E2 -17284.268} C_VEL
LIN {X 0,Y 283.836,Z 589.509,A -85,B 0,C 180,E1 -17287.111,E2 -17287.111} C_VEL
LIN {X 0,Y 284.537,Z 588.648,A -85,B 0,C 180,E1 -17288.554,E2 -17288.554} C_VEL
LIN {X 0,Y 284.508,Z 587.754,A -85,B 0,C 180,E1 -17289.728,E2 -17289.728} C_VEL
LIN {X 0,Y 282.834,Z 586.093,A -85,B 0,C 180,E1 -17291.676,E2 -17291.676} C_VEL
LIN {X 0,Y 281.432,Z 583.931,A -85,B 0,C 180,E1 -17293.617,E2 -17293.617} C_VEL
LIN {X 0,Y 281.817,Z 582.098,A -85,B 0,C 180,E1 -17294.753,E2 -17294.753} C_VEL
LIN {X 0,Y 283.637,Z 578.367,A -85,B 0,C 180,E1 -17296.556,E2 -17296.556} C_VEL
LIN {X 0,Y 286.561,Z 572.074,A -85,B 0,C 180,E1 -17298.963,E2 -17298.963} C_VEL
LIN {X 0,Y 289.595,Z 565.325,A -85,B 0,C 180,E1 -17300.975,E2 -17300.975} C_VEL
LIN {X 0,Y 293.627,Z 555.667,A -85,B 0,C 180,E1 -17303.261,E2 -17303.261} C_VEL
LIN {X 0,Y 297.359,Z 545.567,A -85,B 0,C 180,E1 -17305.177,E2 -17305.177} C_VEL
LIN {X 0,Y 299.087,Z 540.291,A -85,B 0,C 180,E1 -17306.042,E2 -17306.042} C_VEL
LIN {X 0,Y 297.835,Z 532.417,A -85,B 0,C 180,E1 -17308.16,E2 -17308.16} C_VEL
LIN {X 0,Y 295.656,Z 525.243,A -85,B 0,C 180,E1 -17310.405,E2 -17310.405} C_VEL
LIN {X 0,Y 292.953,Z 518.7,A -85,B 0,C 180,E1 -17312.896,E2 -17312.896} C_VEL
LIN {X 0,Y 290.252,Z 513.426,A -85,B 0,C 180,E1 -17315.529,E2 -17315.529} C_VEL
LIN {X 0,Y 289.048,Z 511.996,A -85,B 0,C 180,E1 -17316.642,E2 -17316.642} C_VEL
LIN {X 0,Y 288.504,Z 510.57,A -85,B 0,C 180,E1 -17317.517,E2 -17317.517} C_VEL
LIN {X 0,Y 286.26,Z 508.725,A -85,B 0,C 180,E1 -17320.44,E2 -17320.44} C_VEL
LIN {X 0,Y 285.419,Z 507.802,A -85,B 0,C 180,E1 -17323.587,E2 -17323.587} C_VEL
LIN {X 0,Y 285.45,Z 508.342,A -85,B 0,C 180,E1 -17325.561,E2 -17325.561} C_VEL
LIN {X 0,Y 285.816,Z 510.072,A -85,B 0,C 180,E1 -17327.534,E2 -17327.534} C_VEL
LIN {X 0,Y 287.104,Z 514.393,A -85,B 0,C 180,E1 -17330.472,E2 -17330.472} C_VEL
LIN {X 0,Y 288.317,Z 516.794,A -85,B 0,C 180,E1 -17331.921,E2 -17331.921} C_VEL
LIN {X 0,Y 290.133,Z 523.807,A -85,B 0,C 180,E1 -17334.453,E2 -17334.453} C_VEL
LIN {X 0,Y 291.242,Z 528.39,A -85,B 0,C 180,E1 -17335.832,E2 -17335.832} C_VEL
LIN {X 0,Y 292.838,Z 537.453,A -85,B 0,C 180,E1 -17338.13,E2 -17338.13} C_VEL
LIN {X 0,Y 293.885,Z 546.69,A -85,B 0,C 180,E1 -17340.193,E2 -17340.193} C_VEL
LIN {X 0,Y 294.137,Z 556.263,A -85,B 0,C 180,E1 -17342.136,E2 -17342.136} C_VEL
LIN {X 0,Y 293.238,Z 566.463,A -85,B 0,C 180,E1 -17344.107,E2 -17344.107} C_VEL
LIN {X 0,Y 290.984,Z 575.252,A -85,B 0,C 180,E1 -17345.758,E2 -17345.758} C_VEL
LIN {X 0,Y 287.446,Z 584.965,A -85,B 0,C 180,E1 -17347.73,E2 -17347.73} C_VEL
LIN {X 0,Y 284.318,Z 593.072,A -85,B 0,C 180,E1 -17349.753,E2 -17349.753} C_VEL
LIN {X 0,Y 281.673,Z 599.905,A -85,B 0,C 180,E1 -17351.827,E2 -17351.827} C_VEL
LIN {X 0,Y 279.655,Z 605.6,A -85,B 0,C 180,E1 -17353.952,E2 -17353.952} C_VEL
LIN {X 0,Y 277.402,Z 611.61,A -85,B 0,C 180,E1 -17356.82,E2 -17356.82} C_VEL
LIN {X 0,Y 276.724,Z 614,A -85,B 0,C 180,E1 -17358.277,E2 -17358.277} C_VEL
LIN {X 0,Y 275.736,Z 617.509,A -85,B 0,C 180,E1 -17361.203,E2 -17361.203} C_VEL
LIN {X 0,Y 275.39,Z 619.518,A -85,B 0,C 180,E1 -17364.141,E2 -17364.141} C_VEL
LIN {X 0,Y 275.389,Z 619.925,A -85,B 0,C 180,E1 -17365.609,E2 -17365.609} C_VEL
LIN {X 0,Y 275.636,Z 619.511,A -85,B 0,C 180,E1 -17368.539,E2 -17368.539} C_VEL
LIN {X 0,Y 275.832,Z 618.713,A -85,B 0,C 180,E1 -17370,E2 -17370} C_VEL
LIN {X 0,Y 275.823,Z 617.457,A -85,B 0,C 180,E1 -17371.46,E2 -17371.46} C_VEL
LIN {X 0,Y 275.646,Z 614.668,A -85,B 0,C 180,E1 -17373.654,E2 -17373.654} C_VEL
LIN {X 0,Y 275.785,Z 610.821,A -85,B 0,C 180,E1 -17375.85,E2 -17375.85} C_VEL
LIN {X 0,Y 275.87,Z 605.752,A -85,B 0,C 180,E1 -17378.054,E2 -17378.054} C_VEL
LIN {X 0,Y 276.206,Z 599.346,A -85,B 0,C 180,E1 -17380.26,E2 -17380.26} C_VEL
LIN {X 0,Y 276.901,Z 591.43,A -85,B 0,C 180,E1 -17382.459,E2 -17382.459} C_VEL
LIN {X 0,Y 277.668,Z 583.411,A -85,B 0,C 180,E1 -17384.287,E2 -17384.287} C_VEL
LIN {X 0,Y 278.681,Z 573.712,A -85,B 0,C 180,E1 -17386.105,E2 -17386.105} C_VEL
LIN {X 0,Y 280.014,Z 561.791,A -85,B 0,C 180,E1 -17387.906,E2 -17387.906} C_VEL
LIN {X 0,Y 280.044,Z 557.447,A -85,B 0,C 180,E1 -17388.472,E2 -17388.472} C_VEL
LIN {X 0,Y 278.871,Z 545.038,A -85,B 0,C 180,E1 -17389.89,E2 -17389.89} C_VEL
LIN {X 0,Y 277.502,Z 531.021,A -85,B 0,C 180,E1 -17391.155,E2 -17391.155} C_VEL
LIN {X 0,Y 276.299,Z 516.669,A -85,B 0,C 180,E1 -17392.109,E2 -17392.109} C_VEL
LIN {X 0,Y 276.321,Z 516.018,A -85,B 0,C 180,E1 -17392.181,E2 -17392.181} C_VEL
LIN {X 0,Y 277.234,Z 508.656,A -85,B 0,C 180,E1 -17397.149,E2 -17397.149} C_VEL
LIN {X 0,Y 278.049,Z 503.357,A -85,B 0,C 180,E1 -17400.752,E2 -17400.752} C_VEL
LIN {X 0,Y 279.052,Z 497.882,A -85,B 0,C 180,E1 -17404.517,E2 -17404.517} C_VEL
LIN {X 0,Y 279.397,Z 494.166,A -85,B 0,C 180,E1 -17407.135,E2 -17407.135} C_VEL
LIN {X 0,Y 278.88,Z 490.409,A -85,B 0,C 180,E1 -17409.915,E2 -17409.915} C_VEL
LIN {X 0,Y 277.893,Z 485.152,A -85,B 0,C 180,E1 -17413.956,E2 -17413.956} C_VEL
LIN {X 0,Y 277.4,Z 481.933,A -85,B 0,C 180,E1 -17416.59,E2 -17416.59} C_VEL
LIN {X 0,Y 277.267,Z 481.949,A -85,B 0,C 180,E1 -17420.677,E2 -17420.677} C_VEL
LIN {X 0,Y 277.304,Z 481.941,A -85,B 0,C 180,E1 -17424.344,E2 -17424.344} C_VEL
LIN {X 0,Y 277.244,Z 481.948,A -85,B 0,C 180,E1 -17427.836,E2 -17427.836} C_VEL
LIN {X 0,Y 277.268,Z 481.944,A -85,B 0,C 180,E1 -17431.21,E2 -17431.21} C_VEL
LIN {X 0,Y 277.312,Z 481.942,A -85,B 0,C 180,E1 -17434.48,E2 -17434.48} C_VEL
LIN {X 0,Y 277.287,Z 481.942,A -85,B 0,C 180,E1 -17437.655,E2 -17437.655} C_VEL
LIN {X 0,Y 277.346,Z 481.938,A -85,B 0,C 180,E1 -17440.766,E2 -17440.766} C_VEL
LIN {X 0,Y 277.436,Z 481.924,A -85,B 0,C 180,E1 -17445.326,E2 -17445.326} C_VEL
LIN {X 0,Y 277.508,Z 481.914,A -85,B 0,C 180,E1 -17449.789,E2 -17449.789} C_VEL
LIN {X 0,Y 277.655,Z 481.9,A -85,B 0,C 180,E1 -17452.729,E2 -17452.729} C_VEL
LIN {X 0,Y 277.823,Z 481.879,A -85,B 0,C 180,E1 -17458.551,E2 -17458.551} C_VEL
LIN {X 0,Y 277.823,Z 481.875,A -85,B 0,C 180,E1 -17461.45,E2 -17461.45} C_VEL
LIN {X 0,Y 277.655,Z 481.895,A -85,B 0,C 180,E1 -17467.271,E2 -17467.271} C_VEL
LIN {X 0,Y 277.508,Z 481.918,A -85,B 0,C 180,E1 -17470.212,E2 -17470.212} C_VEL
LIN {X 0,Y 277.436,Z 481.925,A -85,B 0,C 180,E1 -17474.674,E2 -17474.674} C_VEL
LIN {X 0,Y 277.347,Z 481.935,A -85,B 0,C 180,E1 -17479.234,E2 -17479.234} C_VEL
LIN {X 0,Y 277.321,Z 481.94,A -85,B 0,C 180,E1 -17484.171,E2 -17484.171} C_VEL
LIN {X 0,Y 277.328,Z 481.937,A -85,B 0,C 180,E1 -17487.506,E2 -17487.506} C_VEL
LIN {X 0,Y 277.274,Z 481.947,A -85,B 0,C 180,E1 -17490.482,E2 -17490.482} C_VEL
LIN {X 0,Y 277.249,Z 481.947,A -85,B 0,C 180,E1 -17493.896,E2 -17493.896} C_VEL
LIN {X 0,Y 277.274,Z 481.944,A -85,B 0,C 180,E1 -17497.469,E2 -17497.469} C_VEL
LIN {X 0,Y 277.212,Z 481.95,A -85,B 0,C 180,E1 -17501.237,E2 -17501.237} C_VEL
LIN {X 0,Y 277.203,Z 481.953,A -85,B 0,C 180,E1 -17505.227,E2 -17505.227} C_VEL
LIN {X 0,Y 277.225,Z 481.95,A -85,B 0,C 180,E1 -17509.512,E2 -17509.512} C_VEL
LIN {X 0,Y 277.284,Z 481.945,A -85,B 0,C 180,E1 -17512.533,E2 -17512.533} C_VEL
LIN {X 0,Y 277.257,Z 481.95,A -85,B 0,C 180,E1 -17516.106,E2 -17516.106} C_VEL
LIN {X 0,Y 277.264,Z 481.944,A -85,B 0,C 180,E1 -17519.539,E2 -17519.539} C_VEL
LIN {X 0,Y 277.36,Z 481.934,A -85,B 0,C 180,E1 -17522.864,E2 -17522.864} C_VEL
LIN {X 0,Y 277.332,Z 481.941,A -85,B 0,C 180,E1 -17526.08,E2 -17526.08} C_VEL
LIN {X 0,Y 277.348,Z 481.935,A -85,B 0,C 180,E1 -17530.767,E2 -17530.767} C_VEL
LIN {X 0,Y 277.438,Z 481.923,A -85,B 0,C 180,E1 -17535.326,E2 -17535.326} C_VEL
LIN {X 0,Y 277.464,Z 481.923,A -85,B 0,C 180,E1 -17539.787,E2 -17539.787} C_VEL
LIN {X 0,Y 277.616,Z 481.901,A -85,B 0,C 180,E1 -17542.728,E2 -17542.728} C_VEL
LIN {X 0,Y 277.826,Z 481.876,A -85,B 0,C 180,E1 -17548.551,E2 -17548.551} C_VEL
LIN {X 0,Y 277.825,Z 481.876,A -85,B 0,C 180,E1 -17551.45,E2 -17551.45} C_VEL
LIN {X 0,Y 277.645,Z 481.898,A -85,B 0,C 180,E1 -17557.271,E2 -17557.271} C_VEL
LIN {X 0,Y 277.465,Z 481.922,A -85,B 0,C 180,E1 -17560.213,E2 -17560.213} C_VEL
LIN {X 0,Y 277.439,Z 481.923,A -85,B 0,C 180,E1 -17564.674,E2 -17564.674} C_VEL
LIN {X 0,Y 277.349,Z 481.935,A -85,B 0,C 180,E1 -17569.234,E2 -17569.234} C_VEL
LIN {X 0,Y 277.323,Z 481.94,A -85,B 0,C 180,E1 -17574.171,E2 -17574.171} C_VEL
LIN {X 0,Y 277.327,Z 481.939,A -85,B 0,C 180,E1 -17577.504,E2 -17577.504} C_VEL
LIN {X 0,Y 277.275,Z 481.943,A -85,B 0,C 180,E1 -17580.481,E2 -17580.481} C_VEL
LIN {X 0,Y 277.251,Z 481.951,A -85,B 0,C 180,E1 -17583.896,E2 -17583.896} C_VEL
LIN {X 0,Y 277.277,Z 481.946,A -85,B 0,C 180,E1 -17587.468,E2 -17587.468} C_VEL
LIN {X 0,Y 277.213,Z 481.952,A -85,B 0,C 180,E1 -17591.236,E2 -17591.236} C_VEL
LIN {X 0,Y 277.204,Z 481.954,A -85,B 0,C 180,E1 -17595.226,E2 -17595.226} C_VEL
LIN {X 0,Y 277.225,Z 481.952,A -85,B 0,C 180,E1 -17599.512,E2 -17599.512} C_VEL
LIN {X 0,Y 277.202,Z 481.953,A -85,B 0,C 180,E1 -17602.52,E2 -17602.52} C_VEL
LIN {X 0,Y 276.94,Z 481.986,A -85,B 0,C 180,E1 -17606.061,E2 -17606.061} C_VEL
LIN {X 0,Y 276.581,Z 482.034,A -85,B 0,C 180,E1 -17609.763,E2 -17609.763} C_VEL
LIN {X 0,Y 276.249,Z 482.076,A -85,B 0,C 180,E1 -17612.928,E2 -17612.928} C_VEL
LIN {X 0,Y 276.092,Z 482.095,A -85,B 0,C 180,E1 -17614.358,E2 -17614.358} C_VEL
LIN {X 0,Y 275.926,Z 483.139,A -85,B 0,C 180,E1 -17616.484,E2 -17616.484} C_VEL
LIN {X 0,Y 275.895,Z 484.646,A -85,B 0,C 180,E1 -17618.127,E2 -17618.127} C_VEL
LIN {X 0,Y 278.358,Z 498.223,A -85,B 0,C 180,E1 -17619.097,E2 -17619.097} C_VEL
LIN {X 0,Y 280.89,Z 511.723,A -85,B 0,C 180,E1 -17620.353,E2 -17620.353} C_VEL
LIN {X 0,Y 281.719,Z 516.633,A -85,B 0,C 180,E1 -17620.887,E2 -17620.887} C_VEL
LIN {X 0,Y 280.579,Z 528.532,A -85,B 0,C 180,E1 -17622.301,E2 -17622.301} C_VEL
LIN {X 0,Y 279.56,Z 538.541,A -85,B 0,C 180,E1 -17623.759,E2 -17623.759} C_VEL
LIN {X 0,Y 278.598,Z 547.883,A -85,B 0,C 180,E1 -17625.388,E2 -17625.388} C_VEL
LIN {X 0,Y 277.661,Z 556.592,A -85,B 0,C 180,E1 -17627.204,E2 -17627.204} C_VEL
LIN {X 0,Y 276.837,Z 565.228,A -85,B 0,C 180,E1 -17629.394,E2 -17629.394} C_VEL
LIN {X 0,Y 276.171,Z 573.305,A -85,B 0,C 180,E1 -17631.954,E2 -17631.954} C_VEL
LIN {X 0,Y 275.776,Z 578.798,A -85,B 0,C 180,E1 -17634.149,E2 -17634.149} C_VEL
LIN {X 0,Y 275.63,Z 583.114,A -85,B 0,C 180,E1 -17636.345,E2 -17636.345} C_VEL
LIN {X 0,Y 275.503,Z 586.372,A -85,B 0,C 180,E1 -17638.538,E2 -17638.538} C_VEL
LIN {X 0,Y 275.529,Z 588.003,A -85,B 0,C 180,E1 -17640,E2 -17640} C_VEL
LIN {X 0,Y 275.89,Z 590.054,A -85,B 0,C 180,E1 -17642.92,E2 -17642.92} C_VEL
LIN {X 0,Y 276.196,Z 590.506,A -85,B 0,C 180,E1 -17644.378,E2 -17644.378} C_VEL
LIN {X 0,Y 276.837,Z 590.207,A -85,B 0,C 180,E1 -17647.292,E2 -17647.292} C_VEL
LIN {X 0,Y 278.399,Z 588.367,A -85,B 0,C 180,E1 -17650.178,E2 -17650.178} C_VEL
LIN {X 0,Y 280.254,Z 584.968,A -85,B 0,C 180,E1 -17653.044,E2 -17653.044} C_VEL
LIN {X 0,Y 281.817,Z 582.098,A -85,B 0,C 180,E1 -17654.753,E2 -17654.753} C_VEL
LIN {X 0,Y 282.313,Z 580.089,A -85,B 0,C 180,E1 -17655.878,E2 -17655.878} C_VEL
LIN {X 0,Y 281.563,Z 576.825,A -85,B 0,C 180,E1 -17657.777,E2 -17657.777} C_VEL
LIN {X 0,Y 281.081,Z 573.078,A -85,B 0,C 180,E1 -17659.635,E2 -17659.635} C_VEL
LIN {X 0,Y 281.96,Z 570.237,A -85,B 0,C 180,E1 -17660.671,E2 -17660.671} C_VEL
LIN {X 0,Y 285.668,Z 562.609,A -85,B 0,C 180,E1 -17662.798,E2 -17662.798} C_VEL
LIN {X 0,Y 289.399,Z 553.878,A -85,B 0,C 180,E1 -17664.766,E2 -17664.766} C_VEL
LIN {X 0,Y 293.423,Z 543.789,A -85,B 0,C 180,E1 -17666.615,E2 -17666.615} C_VEL
LIN {X 0,Y 293.043,Z 538.912,A -85,B 0,C 180,E1 -17667.957,E2 -17667.957} C_VEL
LIN {X 0,Y 292.292,Z 534.789,A -85,B 0,C 180,E1 -17669.239,E2 -17669.239} C_VEL
LIN {X 0,Y 290.595,Z 528.813,A -85,B 0,C 180,E1 -17671.339,E2 -17671.339} C_VEL
LIN {X 0,Y 288.984,Z 524.475,A -85,B 0,C 180,E1 -17673.142,E2 -17673.142} C_VEL
LIN {X 0,Y 287.382,Z 520.903,A -85,B 0,C 180,E1 -17674.939,E2 -17674.939} C_VEL
LIN {X 0,Y 285.757,Z 518.216,A -85,B 0,C 180,E1 -17676.794,E2 -17676.794} C_VEL
LIN {X 0,Y 284.963,Z 516.571,A -85,B 0,C 180,E1 -17678.066,E2 -17678.066} C_VEL
LIN {X 0,Y 283.554,Z 515.354,A -85,B 0,C 180,E1 -17680.122,E2 -17680.122} C_VEL
LIN {X 0,Y 282.837,Z 514.578,A -85,B 0,C 180,E1 -17682.137,E2 -17682.137} C_VEL
LIN {X 0,Y 282.647,Z 514.372,A -85,B 0,C 180,E1 -17684.124,E2 -17684.124} C_VEL
LIN {X 0,Y 282.747,Z 515.318,A -85,B 0,C 180,E1 -17686.123,E2 -17686.123} C_VEL
LIN {X 0,Y 283.435,Z 518.787,A -85,B 0,C 180,E1 -17689.041,E2 -17689.041} C_VEL
LIN {X 0,Y 284.58,Z 521.982,A -85,B 0,C 180,E1 -17691.092,E2 -17691.092} C_VEL
LIN {X 0,Y 285.297,Z 525.351,A -85,B 0,C 180,E1 -17692.524,E2 -17692.524} C_VEL
LIN {X 0,Y 286.258,Z 529.685,A -85,B 0,C 180,E1 -17694.115,E2 -17694.115} C_VEL
LIN {X 0,Y 287.157,Z 535.041,A -85,B 0,C 180,E1 -17695.742,E2 -17695.742} C_VEL
LIN {X 0,Y 288.172,Z 543.526,A -85,B 0,C 180,E1 -17697.977,E2 -17697.977} C_VEL
LIN {X 0,Y 288.682,Z 552.961,A -85,B 0,C 180,E1 -17700.175,E2 -17700.175} C_VEL
LIN {X 0,Y 288.282,Z 561.698,A -85,B 0,C 180,E1 -17702.044,E2 -17702.044} C_VEL
LIN {X 0,Y 286.861,Z 570.387,A -85,B 0,C 180,E1 -17703.832,E2 -17703.832} C_VEL
LIN {X 0,Y 284.725,Z 577.264,A -85,B 0,C 180,E1 -17705.189,E2 -17705.189} C_VEL
LIN {X 0,Y 280.407,Z 587.794,A -85,B 0,C 180,E1 -17707.529,E2 -17707.529} C_VEL
LIN {X 0,Y 277.164,Z 595.612,A -85,B 0,C 180,E1 -17709.682,E2 -17709.682} C_VEL
LIN {X 0,Y 274.994,Z 600.678,A -85,B 0,C 180,E1 -17711.369,E2 -17711.369} C_VEL
LIN {X 0,Y 272.852,Z 606.095,A -85,B 0,C 180,E1 -17713.541,E2 -17713.541} C_VEL
LIN {X 0,Y 271.015,Z 610.538,A -85,B 0,C 180,E1 -17715.738,E2 -17715.738} C_VEL
LIN {X 0,Y 269.734,Z 614.032,A -85,B 0,C 180,E1 -17717.969,E2 -17717.969} C_VEL
LIN {X 0,Y 268.697,Z 617.357,A -85,B 0,C 180,E1 -17720.971,E2 -17720.971} C_VEL
LIN {X 0,Y 268.409,Z 618.443,A -85,B 0,C 180,E1 -17722.477,E2 -17722.477} C_VEL
LIN {X 0,Y 268.31,Z 619.417,A -85,B 0,C 180,E1 -17725.493,E2 -17725.493} C_VEL
LIN {X 0,Y 268.568,Z 618.841,A -85,B 0,C 180,E1 -17728.5,E2 -17728.5} C_VEL
LIN {X 0,Y 268.779,Z 617.94,A -85,B 0,C 180,E1 -17730,E2 -17730} C_VEL
LIN {X 0,Y 268.769,Z 616.559,A -85,B 0,C 180,E1 -17731.498,E2 -17731.498} C_VEL
LIN {X 0,Y 268.607,Z 613.64,A -85,B 0,C 180,E1 -17733.75,E2 -17733.75} C_VEL
LIN {X 0,Y 268.724,Z 609.625,A -85,B 0,C 180,E1 -17736.005,E2 -17736.005} C_VEL
LIN {X 0,Y 268.891,Z 603.375,A -85,B 0,C 180,E1 -17738.643,E2 -17738.643} C_VEL
LIN {X 0,Y 269.294,Z 596.527,A -85,B 0,C 180,E1 -17740.907,E2 -17740.907} C_VEL
LIN {X 0,Y 270.071,Z 588.017,A -85,B 0,C 180,E1 -17743.162,E2 -17743.162} C_VEL
LIN {X 0,Y 270.933,Z 579.406,A -85,B 0,C 180,E1 -17745.034,E2 -17745.034} C_VEL
LIN {X 0,Y 272.135,Z 568.678,A -85,B 0,C 180,E1 -17746.945,E2 -17746.945} C_VEL
LIN {X 0,Y 273.039,Z 558.818,A -85,B 0,C 180,E1 -17748.38,E2 -17748.38} C_VEL
LIN {X 0,Y 271.815,Z 545.64,A -85,B 0,C 180,E1 -17749.968,E2 -17749.968} C_VEL
LIN {X 0,Y 270.529,Z 532.23,A -85,B 0,C 180,E1 -17751.236,E2 -17751.236} C_VEL
LIN {X 0,Y 269.378,Z 518.459,A -85,B 0,C 180,E1 -17752.228,E2 -17752.228} C_VEL
LIN {X 0,Y 269.267,Z 515.677,A -85,B 0,C 180,E1 -17752.44,E2 -17752.44} C_VEL
LIN {X 0,Y 270.127,Z 509.04,A -85,B 0,C 180,E1 -17757.06,E2 -17757.06} C_VEL
LIN {X 0,Y 271.051,Z 503.09,A -85,B 0,C 180,E1 -17761.237,E2 -17761.237} C_VEL
LIN {X 0,Y 272.213,Z 497.072,A -85,B 0,C 180,E1 -17765.514,E2 -17765.514} C_VEL
LIN {X 0,Y 272.332,Z 495.206,A -85,B 0,C 180,E1 -17766.869,E2 -17766.869} C_VEL
LIN {X 0,Y 271.99,Z 492.129,A -85,B 0,C 180,E1 -17769.179,E2 -17769.179} C_VEL
LIN {X 0,Y 270.978,Z 486.71,A -85,B 0,C 180,E1 -17773.431,E2 -17773.431} C_VEL
LIN {X 0,Y 270.359,Z 482.81,A -85,B 0,C 180,E1 -17776.707,E2 -17776.707} C_VEL
LIN {X 0,Y 270.245,Z 482.819,A -85,B 0,C 180,E1 -17781.381,E2 -17781.381} C_VEL
LIN {X 0,Y 270.215,Z 482.825,A -85,B 0,C 180,E1 -17785.097,E2 -17785.097} C_VEL
LIN {X 0,Y 270.201,Z 482.826,A -85,B 0,C 180,E1 -17789.131,E2 -17789.131} C_VEL
LIN {X 0,Y 270.263,Z 482.817,A -85,B 0,C 180,E1 -17792.146,E2 -17792.146} C_VEL
LIN {X 0,Y 270.278,Z 482.816,A -85,B 0,C 180,E1 -17795.519,E2 -17795.519} C_VEL
LIN {X 0,Y 270.303,Z 482.813,A -85,B 0,C 180,E1 -17800.245,E2 -17800.245} C_VEL
LIN {X 0,Y 270.404,Z 482.802,A -85,B 0,C 180,E1 -17804.936,E2 -17804.936} C_VEL
LIN {X 0,Y 270.443,Z 482.793,A -85,B 0,C 180,E1 -17809.519,E2 -17809.519} C_VEL
LIN {X 0,Y 270.613,Z 482.778,A -85,B 0,C 180,E1 -17812.539,E2 -17812.539} C_VEL
LIN {X 0,Y 270.789,Z 482.755,A -85,B 0,C 180,E1 -17818.513,E2 -17818.513} C_VEL
LIN {X 0,Y 270.789,Z 482.752,A -85,B 0,C 180,E1 -17821.487,E2 -17821.487} C_VEL
LIN {X 0,Y 270.613,Z 482.772,A -85,B 0,C 180,E1 -17827.461,E2 -17827.461} C_VEL
LIN {X 0,Y 270.443,Z 482.799,A -85,B 0,C 180,E1 -17830.481,E2 -17830.481} C_VEL
LIN {X 0,Y 270.405,Z 482.798,A -85,B 0,C 180,E1 -17835.065,E2 -17835.065} C_VEL
LIN {X 0,Y 270.303,Z 482.813,A -85,B 0,C 180,E1 -17839.756,E2 -17839.756} C_VEL
LIN {X 0,Y 270.276,Z 482.818,A -85,B 0,C 180,E1 -17844.586,E2 -17844.586} C_VEL
LIN {X 0,Y 270.274,Z 482.817,A -85,B 0,C 180,E1 -17847.909,E2 -17847.909} C_VEL
LIN {X 0,Y 270.186,Z 482.826,A -85,B 0,C 180,E1 -17851.348,E2 -17851.348} C_VEL
LIN {X 0,Y 270.204,Z 482.825,A -85,B 0,C 180,E1 -17854.906,E2 -17854.906} C_VEL
LIN {X 0,Y 270.199,Z 482.826,A -85,B 0,C 180,E1 -17858.711,E2 -17858.711} C_VEL
LIN {X 0,Y 270.174,Z 482.83,A -85,B 0,C 180,E1 -17862.559,E2 -17862.559} C_VEL
LIN {X 0,Y 270.167,Z 482.83,A -85,B 0,C 180,E1 -17866.751,E2 -17866.751} C_VEL
LIN {X 0,Y 270.225,Z 482.821,A -85,B 0,C 180,E1 -17871.283,E2 -17871.283} C_VEL
LIN {X 0,Y 270.226,Z 482.822,A -85,B 0,C 180,E1 -17875.098,E2 -17875.098} C_VEL
LIN {X 0,Y 270.203,Z 482.823,A -85,B 0,C 180,E1 -17879.131,E2 -17879.131} C_VEL
LIN {X 0,Y 270.266,Z 482.821,A -85,B 0,C 180,E1 -17882.147,E2 -17882.147} C_VEL
LIN {X 0,Y 270.28,Z 482.816,A -85,B 0,C 180,E1 -17885.519,E2 -17885.519} C_VEL
LIN {X 0,Y 270.305,Z 482.816,A -85,B 0,C 180,E1 -17890.245,E2 -17890.245} C_VEL
LIN {X 0,Y 270.407,Z 482.799,A -85,B 0,C 180,E1 -17894.936,E2 -17894.936} C_VEL
LIN {X 0,Y 270.416,Z 482.799,A -85,B 0,C 180,E1 -17899.518,E2 -17899.518} C_VEL
LIN {X 0,Y 270.575,Z 482.779,A -85,B 0,C 180,E1 -17902.538,E2 -17902.538} C_VEL
LIN {X 0,Y 270.791,Z 482.753,A -85,B 0,C 180,E1 -17908.513,E2 -17908.513} C_VEL
LIN {X 0,Y 270.791,Z 482.753,A -85,B 0,C 180,E1 -17911.487,E2 -17911.487} C_VEL
LIN {X 0,Y 270.602,Z 482.776,A -85,B 0,C 180,E1 -17917.462,E2 -17917.462} C_VEL
LIN {X 0,Y 270.417,Z 482.799,A -85,B 0,C 180,E1 -17920.482,E2 -17920.482} C_VEL
LIN {X 0,Y 270.407,Z 482.799,A -85,B 0,C 180,E1 -17925.065,E2 -17925.065} C_VEL
LIN {X 0,Y 270.306,Z 482.816,A -85,B 0,C 180,E1 -17929.755,E2 -17929.755} C_VEL
LIN {X 0,Y 270.278,Z 482.816,A -85,B 0,C 180,E1 -17934.585,E2 -17934.585} C_VEL
LIN {X 0,Y 270.273,Z 482.82,A -85,B 0,C 180,E1 -17937.909,E2 -17937.909} C_VEL
LIN {X 0,Y 270.188,Z 482.826,A -85,B 0,C 180,E1 -17941.348,E2 -17941.348} C_VEL
LIN {X 0,Y 270.206,Z 482.824,A -85,B 0,C 180,E1 -17944.905,E2 -17944.905} C_VEL
LIN {X 0,Y 270.226,Z 482.82,A -85,B 0,C 180,E1 -17948.717,E2 -17948.717} C_VEL
LIN {X 0,Y 270.168,Z 482.83,A -85,B 0,C 180,E1 -17953.249,E2 -17953.249} C_VEL
LIN {X 0,Y 270.175,Z 482.83,A -85,B 0,C 180,E1 -17957.442,E2 -17957.442} C_VEL
LIN {X 0,Y 270.167,Z 482.831,A -85,B 0,C 180,E1 -17961.367,E2 -17961.367} C_VEL
LIN {X 0,Y 269.973,Z 482.854,A -85,B 0,C 180,E1 -17965.06,E2 -17965.06} C_VEL
LIN {X 0,Y 269.625,Z 482.896,A -85,B 0,C 180,E1 -17968.579,E2 -17968.579} C_VEL
LIN {X 0,Y 269.261,Z 482.948,A -85,B 0,C 180,E1 -17972.554,E2 -17972.554} C_VEL
LIN {X 0,Y 268.864,Z 483.196,A -85,B 0,C 180,E1 -17975.812,E2 -17975.812} C_VEL
LIN {X 0,Y 268.803,Z 484.941,A -85,B 0,C 180,E1 -17977.873,E2 -17977.873} C_VEL
LIN {X 0,Y 271.236,Z 498.541,A -85,B 0,C 180,E1 -17978.876,E2 -17978.876} C_VEL
LIN {X 0,Y 273.723,Z 512.063,A -85,B 0,C 180,E1 -17980.172,E2 -17980.172} C_VEL
LIN {X 0,Y 274.65,Z 517.354,A -85,B 0,C 180,E1 -17980.764,E2 -17980.764} C_VEL
LIN {X 0,Y 273.465,Z 529.287,A -85,B 0,C 180,E1 -17982.23,E2 -17982.23} C_VEL
LIN {X 0,Y 272.432,Z 539.132,A -85,B 0,C 180,E1 -17983.707,E2 -17983.707} C_VEL
LIN {X 0,Y 271.481,Z 548.455,A -85,B 0,C 180,E1 -17985.38,E2 -17985.38} C_VEL
LIN {X 0,Y 270.536,Z 557.149,A -85,B 0,C 180,E1 -17987.243,E2 -17987.243} C_VEL
LIN {X 0,Y 269.695,Z 565.766,A -85,B 0,C 180,E1 -17989.489,E2 -17989.489} C_VEL
LIN {X 0,Y 269.052,Z 573.8,A -85,B 0,C 180,E1 -17992.117,E2 -17992.117} C_VEL
LIN {X 0,Y 268.623,Z 580.032,A -85,B 0,C 180,E1 -17994.746,E2 -17994.746} C_VEL
LIN {X 0,Y 268.51,Z 584.168,A -85,B 0,C 180,E1 -17996.999,E2 -17996.999} C_VEL
LIN {X 0,Y 268.442,Z 588.123,A -85,B 0,C 180,E1 -18000,E2 -18000} C_VEL
LIN {X 0,Y 268.579,Z 589.465,A -85,B 0,C 180,E1 -18001.499,E2 -18001.499} C_VEL
LIN {X 0,Y 269.128,Z 590.928,A -85,B 0,C 180,E1 -18004.493,E2 -18004.493} C_VEL
LIN {X 0,Y 269.844,Z 590.907,A -85,B 0,C 180,E1 -18007.482,E2 -18007.482} C_VEL
LIN {X 0,Y 271.485,Z 589.273,A -85,B 0,C 180,E1 -18010.44,E2 -18010.44} C_VEL
LIN {X 0,Y 273.45,Z 586.2,A -85,B 0,C 180,E1 -18013.374,E2 -18013.374} C_VEL
LIN {X 0,Y 276.237,Z 581.41,A -85,B 0,C 180,E1 -18016.252,E2 -18016.252} C_VEL
LIN {X 0,Y 278.758,Z 576.723,A -85,B 0,C 180,E1 -18018.37,E2 -18018.37} C_VEL
LIN {X 0,Y 281.96,Z 570.237,A -85,B 0,C 180,E1 -18020.671,E2 -18020.671} C_VEL
LIN {X 0,Y 282.979,Z 567.27,A -85,B 0,C 180,E1 -18021.691,E2 -18021.691} C_VEL
LIN {X 0,Y 283.237,Z 562.547,A -85,B 0,C 180,E1 -18023.461,E2 -18023.461} C_VEL
LIN {X 0,Y 283.67,Z 557.331,A -85,B 0,C 180,E1 -18025.155,E2 -18025.155} C_VEL
LIN {X 0,Y 284.903,Z 553.603,A -85,B 0,C 180,E1 -18026.036,E2 -18026.036} C_VEL
LIN {X 0,Y 287.581,Z 547.38,A -85,B 0,C 180,E1 -18027.199,E2 -18027.199} C_VEL
LIN {X 0,Y 287.946,Z 545.556,A -85,B 0,C 180,E1 -18027.629,E2 -18027.629} C_VEL
LIN {X 0,Y 287.472,Z 540.424,A -85,B 0,C 180,E1 -18029.272,E2 -18029.272} C_VEL
LIN {X 0,Y 285.988,Z 533.824,A -85,B 0,C 180,E1 -18031.728,E2 -18031.728} C_VEL
LIN {X 0,Y 284.57,Z 529.424,A -85,B 0,C 180,E1 -18033.724,E2 -18033.724} C_VEL
LIN {X 0,Y 282.897,Z 525.365,A -85,B 0,C 180,E1 -18036.066,E2 -18036.066} C_VEL
LIN {X 0,Y 281.234,Z 522.499,A -85,B 0,C 180,E1 -18038.664,E2 -18038.664} C_VEL
LIN {X 0,Y 280.002,Z 521.314,A -85,B 0,C 180,E1 -18041.149,E2 -18041.149} C_VEL
LIN {X 0,Y 279.641,Z 520.845,A -85,B 0,C 180,E1 -18043.211,E2 -18043.211} C_VEL
LIN {X 0,Y 279.642,Z 521.324,A -85,B 0,C 180,E1 -18045.275,E2 -18045.275} C_VEL
LIN {X 0,Y 279.809,Z 523.081,A -85,B 0,C 180,E1 -18047.299,E2 -18047.299} C_VEL
LIN {X 0,Y 280.483,Z 526.401,A -85,B 0,C 180,E1 -18049.741,E2 -18049.741} C_VEL
LIN {X 0,Y 281.298,Z 529.147,A -85,B 0,C 180,E1 -18051.346,E2 -18051.346} C_VEL
LIN {X 0,Y 282.057,Z 533.882,A -85,B 0,C 180,E1 -18053.272,E2 -18053.272} C_VEL
LIN {X 0,Y 282.658,Z 539.623,A -85,B 0,C 180,E1 -18055.136,E2 -18055.136} C_VEL
LIN {X 0,Y 283.248,Z 548.15,A -85,B 0,C 180,E1 -18057.524,E2 -18057.524} C_VEL
LIN {X 0,Y 283.267,Z 556.481,A -85,B 0,C 180,E1 -18059.591,E2 -18059.591} C_VEL
LIN {X 0,Y 282.506,Z 564.631,A -85,B 0,C 180,E1 -18061.464,E2 -18061.464} C_VEL
LIN {X 0,Y 280.852,Z 572.747,A -85,B 0,C 180,E1 -18063.228,E2 -18063.228} C_VEL
LIN {X 0,Y 277.789,Z 580.732,A -85,B 0,C 180,E1 -18064.927,E2 -18064.927} C_VEL
LIN {X 0,Y 273.383,Z 590.524,A -85,B 0,C 180,E1 -18067.318,E2 -18067.318} C_VEL
LIN {X 0,Y 269.935,Z 597.936,A -85,B 0,C 180,E1 -18069.602,E2 -18069.602} C_VEL
LIN {X 0,Y 266.773,Z 605,A -85,B 0,C 180,E1 -18072.364,E2 -18072.364} C_VEL
LIN {X 0,Y 264.15,Z 610.825,A -85,B 0,C 180,E1 -18075.359,E2 -18075.359} C_VEL
LIN {X 0,Y 262.754,Z 614.115,A -85,B 0,C 180,E1 -18077.644,E2 -18077.644} C_VEL
LIN {X 0,Y 261.674,Z 617.159,A -85,B 0,C 180,E1 -18080.726,E2 -18080.726} C_VEL
LIN {X 0,Y 261.226,Z 618.696,A -85,B 0,C 180,E1 -18083.822,E2 -18083.822} C_VEL
LIN {X 0,Y 261.233,Z 618.903,A -85,B 0,C 180,E1 -18085.37,E2 -18085.37} C_VEL
LIN {X 0,Y 261.278,Z 618.722,A -85,B 0,C 180,E1 -18086.916,E2 -18086.916} C_VEL
LIN {X 0,Y 261.502,Z 618.125,A -85,B 0,C 180,E1 -18088.46,E2 -18088.46} C_VEL
LIN {X 0,Y 261.727,Z 617.102,A -85,B 0,C 180,E1 -18090,E2 -18090} C_VEL
LIN {X 0,Y 261.716,Z 615.634,A -85,B 0,C 180,E1 -18091.539,E2 -18091.539} C_VEL
LIN {X 0,Y 261.589,Z 612.538,A -85,B 0,C 180,E1 -18093.851,E2 -18093.851} C_VEL
LIN {X 0,Y 261.726,Z 607.653,A -85,B 0,C 180,E1 -18096.514,E2 -18096.514} C_VEL
LIN {X 0,Y 261.892,Z 601.918,A -85,B 0,C 180,E1 -18098.876,E2 -18098.876} C_VEL
LIN {X 0,Y 262.316,Z 594.831,A -85,B 0,C 180,E1 -18101.2,E2 -18101.2} C_VEL
LIN {X 0,Y 263.141,Z 586.086,A -85,B 0,C 180,E1 -18103.515,E2 -18103.515} C_VEL
LIN {X 0,Y 264.146,Z 576.149,A -85,B 0,C 180,E1 -18105.628,E2 -18105.628} C_VEL
LIN {X 0,Y 265.479,Z 564.951,A -85,B 0,C 180,E1 -18107.561,E2 -18107.561} C_VEL
LIN {X 0,Y 265.907,Z 558.519,A -85,B 0,C 180,E1 -18108.491,E2 -18108.491} C_VEL
LIN {X 0,Y 264.783,Z 546.638,A -85,B 0,C 180,E1 -18109.982,E2 -18109.982} C_VEL
LIN {X 0,Y 263.569,Z 533.774,A -85,B 0,C 180,E1 -18111.283,E2 -18111.283} C_VEL
LIN {X 0,Y 262.377,Z 519.493,A -85,B 0,C 180,E1 -18112.387,E2 -18112.387} C_VEL
LIN {X 0,Y 262.226,Z 515.361,A -85,B 0,C 180,E1 -18112.66,E2 -18112.66} C_VEL
LIN {X 0,Y 263.029,Z 509.311,A -85,B 0,C 180,E1 -18117.015,E2 -18117.015} C_VEL
LIN {X 0,Y 263.777,Z 504.609,A -85,B 0,C 180,E1 -18120.413,E2 -18120.413} C_VEL
LIN {X 0,Y 264.933,Z 498.768,A -85,B 0,C 180,E1 -18124.679,E2 -18124.679} C_VEL
LIN {X 0,Y 265.268,Z 496.333,A -85,B 0,C 180,E1 -18126.49,E2 -18126.49} C_VEL
LIN {X 0,Y 264.807,Z 492.225,A -85,B 0,C 180,E1 -18129.676,E2 -18129.676} C_VEL
LIN {X 0,Y 263.796,Z 486.872,A -85,B 0,C 180,E1 -18134.001,E2 -18134.001} C_VEL
LIN {X 0,Y 263.309,Z 483.688,A -85,B 0,C 180,E1 -18136.846,E2 -18136.846} C_VEL
LIN {X 0,Y 263.189,Z 483.698,A -85,B 0,C 180,E1 -18142.108,E2 -18142.108} C_VEL
LIN {X 0,Y 263.184,Z 483.699,A -85,B 0,C 180,E1 -18145.89,E2 -18145.89} C_VEL
LIN {X 0,Y 263.141,Z 483.704,A -85,B 0,C 180,E1 -18149.506,E2 -18149.506} C_VEL
LIN {X 0,Y 263.192,Z 483.7,A -85,B 0,C 180,E1 -18153.003,E2 -18153.003} C_VEL
LIN {X 0,Y 263.185,Z 483.702,A -85,B 0,C 180,E1 -18156.387,E2 -18156.387} C_VEL
LIN {X 0,Y 263.264,Z 483.687,A -85,B 0,C 180,E1 -18159.694,E2 -18159.694} C_VEL
LIN {X 0,Y 263.352,Z 483.682,A -85,B 0,C 180,E1 -18164.522,E2 -18164.522} C_VEL
LIN {X 0,Y 263.375,Z 483.674,A -85,B 0,C 180,E1 -18169.235,E2 -18169.235} C_VEL
LIN {X 0,Y 263.574,Z 483.653,A -85,B 0,C 180,E1 -18172.339,E2 -18172.339} C_VEL
LIN {X 0,Y 263.753,Z 483.631,A -85,B 0,C 180,E1 -18178.473,E2 -18178.473} C_VEL
LIN {X 0,Y 263.754,Z 483.628,A -85,B 0,C 180,E1 -18181.527,E2 -18181.527} C_VEL
LIN {X 0,Y 263.575,Z 483.649,A -85,B 0,C 180,E1 -18187.662,E2 -18187.662} C_VEL
LIN {X 0,Y 263.376,Z 483.678,A -85,B 0,C 180,E1 -18190.766,E2 -18190.766} C_VEL
LIN {X 0,Y 263.353,Z 483.676,A -85,B 0,C 180,E1 -18195.478,E2 -18195.478} C_VEL
LIN {X 0,Y 263.265,Z 483.693,A -85,B 0,C 180,E1 -18200.307,E2 -18200.307} C_VEL
LIN {X 0,Y 263.21,Z 483.695,A -85,B 0,C 180,E1 -18205.292,E2 -18205.292} C_VEL
LIN {X 0,Y 263.182,Z 483.701,A -85,B 0,C 180,E1 -18208.73,E2 -18208.73} C_VEL
LIN {X 0,Y 263.135,Z 483.708,A -85,B 0,C 180,E1 -18212.288,E2 -18212.288} C_VEL
LIN {X 0,Y 263.166,Z 483.703,A -85,B 0,C 180,E1 -18215.982,E2 -18215.982} C_VEL
LIN {X 0,Y 263.107,Z 483.71,A -85,B 0,C 180,E1 -18219.873,E2 -18219.873} C_VEL
LIN {X 0,Y 263.125,Z 483.708,A -85,B 0,C 180,E1 -18223.984,E2 -18223.984} C_VEL
LIN {X 0,Y 263.126,Z 483.708,A -85,B 0,C 180,E1 -18228.407,E2 -18228.407} C_VEL
LIN {X 0,Y 263.168,Z 483.703,A -85,B 0,C 180,E1 -18232.105,E2 -18232.105} C_VEL
LIN {X 0,Y 263.186,Z 483.701,A -85,B 0,C 180,E1 -18235.891,E2 -18235.891} C_VEL
LIN {X 0,Y 263.15,Z 483.702,A -85,B 0,C 180,E1 -18239.507,E2 -18239.507} C_VEL
LIN {X 0,Y 263.194,Z 483.698,A -85,B 0,C 180,E1 -18243.003,E2 -18243.003} C_VEL
LIN {X 0,Y 263.188,Z 483.7,A -85,B 0,C 180,E1 -18246.387,E2 -18246.387} C_VEL
LIN {X 0,Y 263.267,Z 483.689,A -85,B 0,C 180,E1 -18249.694,E2 -18249.694} C_VEL
LIN {X 0,Y 263.355,Z 483.679,A -85,B 0,C 180,E1 -18254.522,E2 -18254.522} C_VEL
LIN {X 0,Y 263.358,Z 483.677,A -85,B 0,C 180,E1 -18259.234,E2 -18259.234} C_VEL
LIN {X 0,Y 263.537,Z 483.657,A -85,B 0,C 180,E1 -18262.338,E2 -18262.338} C_VEL
LIN {X 0,Y 263.755,Z 483.629,A -85,B 0,C 180,E1 -18268.473,E2 -18268.473} C_VEL
LIN {X 0,Y 263.755,Z 483.629,A -85,B 0,C 180,E1 -18271.527,E2 -18271.527} C_VEL
LIN {X 0,Y 263.562,Z 483.654,A -85,B 0,C 180,E1 -18277.662,E2 -18277.662} C_VEL
LIN {X 0,Y 263.359,Z 483.677,A -85,B 0,C 180,E1 -18280.766,E2 -18280.766} C_VEL
LIN {X 0,Y 263.355,Z 483.679,A -85,B 0,C 180,E1 -18285.478,E2 -18285.478} C_VEL
LIN {X 0,Y 263.268,Z 483.689,A -85,B 0,C 180,E1 -18290.307,E2 -18290.307} C_VEL
LIN {X 0,Y 263.212,Z 483.696,A -85,B 0,C 180,E1 -18295.291,E2 -18295.291} C_VEL
LIN {X 0,Y 263.179,Z 483.699,A -85,B 0,C 180,E1 -18298.73,E2 -18298.73} C_VEL
LIN {X 0,Y 263.136,Z 483.706,A -85,B 0,C 180,E1 -18302.288,E2 -18302.288} C_VEL
LIN {X 0,Y 263.18,Z 483.703,A -85,B 0,C 180,E1 -18305.979,E2 -18305.979} C_VEL
LIN {X 0,Y 263.119,Z 483.71,A -85,B 0,C 180,E1 -18309.87,E2 -18309.87} C_VEL
LIN {X 0,Y 263.126,Z 483.709,A -85,B 0,C 180,E1 -18313.984,E2 -18313.984} C_VEL
LIN {X 0,Y 263.127,Z 483.705,A -85,B 0,C 180,E1 -18318.406,E2 -18318.406} C_VEL
LIN {X 0,Y 263.061,Z 483.716,A -85,B 0,C 180,E1 -18322.086,E2 -18322.086} C_VEL
LIN {X 0,Y 262.851,Z 483.741,A -85,B 0,C 180,E1 -18325.983,E2 -18325.983} C_VEL
LIN {X 0,Y 262.548,Z 483.78,A -85,B 0,C 180,E1 -18329.429,E2 -18329.429} C_VEL
LIN {X 0,Y 262.173,Z 483.829,A -85,B 0,C 180,E1 -18332.889,E2 -18332.889} C_VEL
LIN {X 0,Y 261.812,Z 483.884,A -85,B 0,C 180,E1 -18335.88,E2 -18335.88} C_VEL
LIN {X 0,Y 261.754,Z 485.313,A -85,B 0,C 180,E1 -18337.608,E2 -18337.608} C_VEL
LIN {X 0,Y 264.12,Z 498.838,A -85,B 0,C 180,E1 -18338.642,E2 -18338.642} C_VEL
LIN {X 0,Y 266.76,Z 513.229,A -85,B 0,C 180,E1 -18340.071,E2 -18340.071} C_VEL
LIN {X 0,Y 267.59,Z 518.073,A -85,B 0,C 180,E1 -18340.635,E2 -18340.635} C_VEL
LIN {X 0,Y 266.287,Z 531.291,A -85,B 0,C 180,E1 -18342.335,E2 -18342.335} C_VEL
LIN {X 0,Y 265.151,Z 541.983,A -85,B 0,C 180,E1 -18344.038,E2 -18344.038} C_VEL
LIN {X 0,Y 263.901,Z 552.607,A -85,B 0,C 180,E1 -18346.132,E2 -18346.132} C_VEL
LIN {X 0,Y 262.951,Z 562.13,A -85,B 0,C 180,E1 -18348.436,E2 -18348.436} C_VEL
LIN {X 0,Y 262.216,Z 569.848,A -85,B 0,C 180,E1 -18350.746,E2 -18350.746} C_VEL
LIN {X 0,Y 261.766,Z 576.161,A -85,B 0,C 180,E1 -18353.061,E2 -18353.061} C_VEL
LIN {X 0,Y 261.509,Z 581.241,A -85,B 0,C 180,E1 -18355.375,E2 -18355.375} C_VEL
LIN {X 0,Y 261.372,Z 585.217,A -85,B 0,C 180,E1 -18357.688,E2 -18357.688} C_VEL
LIN {X 0,Y 261.358,Z 588.164,A -85,B 0,C 180,E1 -18360,E2 -18360} C_VEL
LIN {X 0,Y 261.738,Z 590.699,A -85,B 0,C 180,E1 -18363.078,E2 -18363.078} C_VEL
LIN {X 0,Y 262.065,Z 591.347,A -85,B 0,C 180,E1 -18364.614,E2 -18364.614} C_VEL
LIN {X 0,Y 262.854,Z 591.539,A -85,B 0,C 180,E1 -18367.682,E2 -18367.682} C_VEL
LIN {X 0,Y 264.576,Z 590.209,A -85,B 0,C 180,E1 -18370.716,E2 -18370.716} C_VEL
LIN {X 0,Y 266.647,Z 587.357,A -85,B 0,C 180,E1 -18373.722,E2 -18373.722} C_VEL
LIN {X 0,Y 268.859,Z 584.188,A -85,B 0,C 180,E1 -18375.93,E2 -18375.93} C_VEL
LIN {X 0,Y 271.303,Z 580.089,A -85,B 0,C 180,E1 -18378.111,E2 -18378.111} C_VEL
LIN {X 0,Y 275.251,Z 573.086,A -85,B 0,C 180,E1 -18380.944,E2 -18380.944} C_VEL
LIN {X 0,Y 279.461,Z 565.133,A -85,B 0,C 180,E1 -18383.334,E2 -18383.334} C_VEL
LIN {X 0,Y 283.389,Z 556.986,A -85,B 0,C 180,E1 -18385.328,E2 -18385.328} C_VEL
LIN {X 0,Y 284.903,Z 553.603,A -85,B 0,C 180,E1 -18386.036,E2 -18386.036} C_VEL
LIN {X 0,Y 285.683,Z 551.116,A -85,B 0,C 180,E1 -18386.619,E2 -18386.619} C_VEL
LIN {X 0,Y 285.651,Z 548.011,A -85,B 0,C 180,E1 -18387.626,E2 -18387.626} C_VEL
LIN {X 0,Y 284.705,Z 545.542,A -85,B 0,C 180,E1 -18388.704,E2 -18388.704} C_VEL
LIN {X 0,Y 281.984,Z 541.16,A -85,B 0,C 180,E1 -18391.023,E2 -18391.023} C_VEL
LIN {X 0,Y 281.41,Z 539.503,A -85,B 0,C 180,E1 -18391.796,E2 -18391.796} C_VEL
LIN {X 0,Y 280.178,Z 534.648,A -85,B 0,C 180,E1 -18394.129,E2 -18394.129} C_VEL
LIN {X 0,Y 278.98,Z 531.191,A -85,B 0,C 180,E1 -18396.279,E2 -18396.279} C_VEL
LIN {X 0,Y 277.813,Z 528.985,A -85,B 0,C 180,E1 -18398.35,E2 -18398.35} C_VEL
LIN {X 0,Y 276.59,Z 527.5,A -85,B 0,C 180,E1 -18401.349,E2 -18401.349} C_VEL
LIN {X 0,Y 276.321,Z 527.153,A -85,B 0,C 180,E1 -18403.371,E2 -18403.371} C_VEL
LIN {X 0,Y 276.308,Z 527.297,A -85,B 0,C 180,E1 -18404.586,E2 -18404.586} C_VEL
LIN {X 0,Y 276.351,Z 528.722,A -85,B 0,C 180,E1 -18406.634,E2 -18406.634} C_VEL
LIN {X 0,Y 276.918,Z 532.539,A -85,B 0,C 180,E1 -18409.586,E2 -18409.586} C_VEL
LIN {X 0,Y 277.33,Z 534.242,A -85,B 0,C 180,E1 -18410.688,E2 -18410.688} C_VEL
LIN {X 0,Y 277.781,Z 538.632,A -85,B 0,C 180,E1 -18412.611,E2 -18412.611} C_VEL
LIN {X 0,Y 278.11,Z 545.121,A -85,B 0,C 180,E1 -18414.843,E2 -18414.843} C_VEL
LIN {X 0,Y 278.175,Z 553.099,A -85,B 0,C 180,E1 -18417.191,E2 -18417.191} C_VEL
LIN {X 0,Y 277.629,Z 561.583,A -85,B 0,C 180,E1 -18419.394,E2 -18419.394} C_VEL
LIN {X 0,Y 276.516,Z 568.73,A -85,B 0,C 180,E1 -18421.124,E2 -18421.124} C_VEL
LIN {X 0,Y 274.827,Z 575.025,A -85,B 0,C 180,E1 -18422.593,E2 -18422.593} C_VEL
LIN {X 0,Y 271.549,Z 582.662,A -85,B 0,C 180,E1 -18424.309,E2 -18424.309} C_VEL
LIN {X 0,Y 266.942,Z 591.833,A -85,B 0,C 180,E1 -18426.739,E2 -18426.739} C_VEL
LIN {X 0,Y 263.518,Z 598.646,A -85,B 0,C 180,E1 -18428.979,E2 -18428.979} C_VEL
LIN {X 0,Y 260.053,Z 605.606,A -85,B 0,C 180,E1 -18431.893,E2 -18431.893} C_VEL
LIN {X 0,Y 257.297,Z 611.066,A -85,B 0,C 180,E1 -18434.96,E2 -18434.96} C_VEL
LIN {X 0,Y 255.783,Z 614.144,A -85,B 0,C 180,E1 -18437.302,E2 -18437.302} C_VEL
LIN {X 0,Y 254.632,Z 616.938,A -85,B 0,C 180,E1 -18440.467,E2 -18440.467} C_VEL
LIN {X 0,Y 254.152,Z 618.275,A -85,B 0,C 180,E1 -18443.649,E2 -18443.649} C_VEL
LIN {X 0,Y 254.16,Z 618.352,A -85,B 0,C 180,E1 -18445.241,E2 -18445.241} C_VEL
LIN {X 0,Y 254.458,Z 617.338,A -85,B 0,C 180,E1 -18448.417,E2 -18448.417} C_VEL
LIN {X 0,Y 254.675,Z 616.245,A -85,B 0,C 180,E1 -18450,E2 -18450} C_VEL
LIN {X 0,Y 254.564,Z 613.699,A -85,B 0,C 180,E1 -18452.373,E2 -18452.373} C_VEL
LIN {X 0,Y 254.58,Z 610.073,A -85,B 0,C 180,E1 -18454.75,E2 -18454.75} C_VEL
LIN {X 0,Y 254.704,Z 605.469,A -85,B 0,C 180,E1 -18457.053,E2 -18457.053} C_VEL
LIN {X 0,Y 254.948,Z 599.216,A -85,B 0,C 180,E1 -18459.52,E2 -18459.52} C_VEL
LIN {X 0,Y 255.509,Z 591.625,A -85,B 0,C 180,E1 -18461.905,E2 -18461.905} C_VEL
LIN {X 0,Y 256.399,Z 582.27,A -85,B 0,C 180,E1 -18464.282,E2 -18464.282} C_VEL
LIN {X 0,Y 257.584,Z 571.691,A -85,B 0,C 180,E1 -18466.444,E2 -18466.444} C_VEL
LIN {X 0,Y 258.85,Z 560.456,A -85,B 0,C 180,E1 -18468.287,E2 -18468.287} C_VEL
LIN {X 0,Y 258.028,Z 550.111,A -85,B 0,C 180,E1 -18469.698,E2 -18469.698} C_VEL
LIN {X 0,Y 256.783,Z 536.93,A -85,B 0,C 180,E1 -18471.162,E2 -18471.162} C_VEL
LIN {X 0,Y 255.666,Z 524.323,A -85,B 0,C 180,E1 -18472.271,E2 -18472.271} C_VEL
LIN {X 0,Y 255.156,Z 515.043,A -85,B 0,C 180,E1 -18472.896,E2 -18472.896} C_VEL
LIN {X 0,Y 256.077,Z 508.439,A -85,B 0,C 180,E1 -18477.811,E2 -18477.811} C_VEL
LIN {X 0,Y 257.089,Z 502.763,A -85,B 0,C 180,E1 -18482.065,E2 -18482.065} C_VEL
LIN {X 0,Y 258.114,Z 497.689,A -85,B 0,C 180,E1 -18485.907,E2 -18485.907} C_VEL
LIN {X 0,Y 257.921,Z 493.999,A -85,B 0,C 180,E1 -18488.808,E2 -18488.808} C_VEL
LIN {X 0,Y 256.955,Z 488.735,A -85,B 0,C 180,E1 -18493.139,E2 -18493.139} C_VEL
LIN {X 0,Y 256.268,Z 484.564,A -85,B 0,C 180,E1 -18496.87,E2 -18496.87} C_VEL
LIN {X 0,Y 256.11,Z 484.582,A -85,B 0,C 180,E1 -18500.865,E2 -18500.865} C_VEL
LIN {X 0,Y 256.121,Z 484.582,A -85,B 0,C 180,E1 -18504.813,E2 -18504.813} C_VEL
LIN {X 0,Y 256.093,Z 484.586,A -85,B 0,C 180,E1 -18508.573,E2 -18508.573} C_VEL
LIN {X 0,Y 256.138,Z 484.576,A -85,B 0,C 180,E1 -18512.196,E2 -18512.196} C_VEL
LIN {X 0,Y 256.168,Z 484.573,A -85,B 0,C 180,E1 -18515.699,E2 -18515.699} C_VEL
LIN {X 0,Y 256.168,Z 484.572,A -85,B 0,C 180,E1 -18519.105,E2 -18519.105} C_VEL
LIN {X 0,Y 256.301,Z 484.558,A -85,B 0,C 180,E1 -18524.085,E2 -18524.085} C_VEL
LIN {X 0,Y 256.311,Z 484.555,A -85,B 0,C 180,E1 -18528.934,E2 -18528.934} C_VEL
LIN {X 0,Y 256.542,Z 484.528,A -85,B 0,C 180,E1 -18532.127,E2 -18532.127} C_VEL
LIN {X 0,Y 256.716,Z 484.507,A -85,B 0,C 180,E1 -18538.432,E2 -18538.432} C_VEL
LIN {X 0,Y 256.716,Z 484.505,A -85,B 0,C 180,E1 -18541.569,E2 -18541.569} C_VEL
LIN {X 0,Y 256.542,Z 484.526,A -85,B 0,C 180,E1 -18547.873,E2 -18547.873} C_VEL
LIN {X 0,Y 256.311,Z 484.556,A -85,B 0,C 180,E1 -18551.066,E2 -18551.066} C_VEL
LIN {X 0,Y 256.302,Z 484.555,A -85,B 0,C 180,E1 -18555.915,E2 -18555.915} C_VEL
LIN {X 0,Y 256.169,Z 484.574,A -85,B 0,C 180,E1 -18560.895,E2 -18560.895} C_VEL
LIN {X 0,Y 256.19,Z 484.569,A -85,B 0,C 180,E1 -18565.139,E2 -18565.139} C_VEL
LIN {X 0,Y 256.116,Z 484.58,A -85,B 0,C 180,E1 -18569.6,E2 -18569.6} C_VEL
LIN {X 0,Y 256.078,Z 484.582,A -85,B 0,C 180,E1 -18573.292,E2 -18573.292} C_VEL
LIN {X 0,Y 256.118,Z 484.579,A -85,B 0,C 180,E1 -18577.272,E2 -18577.272} C_VEL
LIN {X 0,Y 256.056,Z 484.585,A -85,B 0,C 180,E1 -18581.204,E2 -18581.204} C_VEL
LIN {X 0,Y 256.06,Z 484.587,A -85,B 0,C 180,E1 -18585.531,E2 -18585.531} C_VEL
LIN {X 0,Y 256.059,Z 484.586,A -85,B 0,C 180,E1 -18588.797,E2 -18588.797} C_VEL
LIN {X 0,Y 256.147,Z 484.576,A -85,B 0,C 180,E1 -18592.87,E2 -18592.87} C_VEL
LIN {X 0,Y 256.088,Z 484.584,A -85,B 0,C 180,E1 -18596.71,E2 -18596.71} C_VEL
LIN {X 0,Y 256.137,Z 484.576,A -85,B 0,C 180,E1 -18601.407,E2 -18601.407} C_VEL
LIN {X 0,Y 256.17,Z 484.574,A -85,B 0,C 180,E1 -18605.7,E2 -18605.7} C_VEL
LIN {X 0,Y 256.17,Z 484.571,A -85,B 0,C 180,E1 -18609.105,E2 -18609.105} C_VEL
LIN {X 0,Y 256.304,Z 484.56,A -85,B 0,C 180,E1 -18614.085,E2 -18614.085} C_VEL
LIN {X 0,Y 256.299,Z 484.555,A -85,B 0,C 180,E1 -18617.328,E2 -18617.328} C_VEL
LIN {X 0,Y 256.499,Z 484.535,A -85,B 0,C 180,E1 -18622.126,E2 -18622.126} C_VEL
LIN {X 0,Y 256.5,Z 484.531,A -85,B 0,C 180,E1 -18626.859,E2 -18626.859} C_VEL
LIN {X 0,Y 256.769,Z 484.503,A -85,B 0,C 180,E1 -18630,E2 -18630} C_VEL
LIN {X 0,Y 256.502,Z 484.53,A -85,B 0,C 180,E1 -18633.141,E2 -18633.141} C_VEL
LIN {X 0,Y 256.519,Z 484.533,A -85,B 0,C 180,E1 -18637.874,E2 -18637.874} C_VEL
LIN {X 0,Y 256.299,Z 484.555,A -85,B 0,C 180,E1 -18642.672,E2 -18642.672} C_VEL
LIN {X 0,Y 256.287,Z 484.56,A -85,B 0,C 180,E1 -18646.302,E2 -18646.302} C_VEL
LIN {X 0,Y 256.161,Z 484.573,A -85,B 0,C 180,E1 -18651.12,E2 -18651.12} C_VEL
LIN {X 0,Y 256.192,Z 484.57,A -85,B 0,C 180,E1 -18655.139,E2 -18655.139} C_VEL
LIN {X 0,Y 256.114,Z 484.582,A -85,B 0,C 180,E1 -18659.6,E2 -18659.6} C_VEL
LIN {X 0,Y 256.08,Z 484.585,A -85,B 0,C 180,E1 -18663.291,E2 -18663.291} C_VEL
LIN {X 0,Y 256.126,Z 484.579,A -85,B 0,C 180,E1 -18667.273,E2 -18667.273} C_VEL
LIN {X 0,Y 256.06,Z 484.586,A -85,B 0,C 180,E1 -18671.203,E2 -18671.203} C_VEL
LIN {X 0,Y 256.061,Z 484.589,A -85,B 0,C 180,E1 -18675.53,E2 -18675.53} C_VEL
LIN {X 0,Y 256.055,Z 484.585,A -85,B 0,C 180,E1 -18678.796,E2 -18678.796} C_VEL
LIN {X 0,Y 255.997,Z 484.595,A -85,B 0,C 180,E1 -18682.844,E2 -18682.844} C_VEL
LIN {X 0,Y 255.721,Z 484.627,A -85,B 0,C 180,E1 -18686.656,E2 -18686.656} C_VEL
LIN {X 0,Y 255.369,Z 484.673,A -85,B 0,C 180,E1 -18690.305,E2 -18690.305} C_VEL
LIN {X 0,Y 254.99,Z 484.723,A -85,B 0,C 180,E1 -18693.832,E2 -18693.832} C_VEL
LIN {X 0,Y 254.704,Z 484.936,A -85,B 0,C 180,E1 -18696.415,E2 -18696.415} C_VEL
LIN {X 0,Y 254.698,Z 485.878,A -85,B 0,C 180,E1 -18697.392,E2 -18697.392} C_VEL
LIN {X 0,Y 256.978,Z 499.036,A -85,B 0,C 180,E1 -18698.413,E2 -18698.413} C_VEL
LIN {X 0,Y 259.48,Z 512.755,A -85,B 0,C 180,E1 -18699.797,E2 -18699.797} C_VEL
LIN {X 0,Y 260.518,Z 518.675,A -85,B 0,C 180,E1 -18700.498,E2 -18700.498} C_VEL
LIN {X 0,Y 259.26,Z 530.937,A -85,B 0,C 180,E1 -18702.124,E2 -18702.124} C_VEL
LIN {X 0,Y 258.064,Z 542.357,A -85,B 0,C 180,E1 -18703.994,E2 -18703.994} C_VEL
LIN {X 0,Y 256.775,Z 552.966,A -85,B 0,C 180,E1 -18706.143,E2 -18706.143} C_VEL
LIN {X 0,Y 255.798,Z 562.512,A -85,B 0,C 180,E1 -18708.51,E2 -18708.51} C_VEL
LIN {X 0,Y 255.083,Z 570.255,A -85,B 0,C 180,E1 -18710.884,E2 -18710.884} C_VEL
LIN {X 0,Y 254.706,Z 575.638,A -85,B 0,C 180,E1 -18712.867,E2 -18712.867} C_VEL
LIN {X 0,Y 254.415,Z 580.886,A -85,B 0,C 180,E1 -18715.246,E2 -18715.246} C_VEL
LIN {X 0,Y 254.301,Z 585.035,A -85,B 0,C 180,E1 -18717.624,E2 -18717.624} C_VEL
LIN {X 0,Y 254.277,Z 588.188,A -85,B 0,C 180,E1 -18720,E2 -18720} C_VEL
LIN {X 0,Y 254.666,Z 590.932,A -85,B 0,C 180,E1 -18723.164,E2 -18723.164} C_VEL
LIN {X 0,Y 255.005,Z 591.731,A -85,B 0,C 180,E1 -18724.742,E2 -18724.742} C_VEL
LIN {X 0,Y 255.869,Z 592.167,A -85,B 0,C 180,E1 -18727.893,E2 -18727.893} C_VEL
LIN {X 0,Y 257.653,Z 591.081,A -85,B 0,C 180,E1 -18731.007,E2 -18731.007} C_VEL
LIN {X 0,Y 258.662,Z 590.027,A -85,B 0,C 180,E1 -18732.554,E2 -18732.554} C_VEL
LIN {X 0,Y 259.881,Z 588.564,A -85,B 0,C 180,E1 -18734.086,E2 -18734.086} C_VEL
LIN {X 0,Y 262.948,Z 584.438,A -85,B 0,C 180,E1 -18737.098,E2 -18737.098} C_VEL
LIN {X 0,Y 265.771,Z 580.299,A -85,B 0,C 180,E1 -18739.302,E2 -18739.302} C_VEL
LIN {X 0,Y 268.884,Z 575.161,A -85,B 0,C 180,E1 -18741.465,E2 -18741.465} C_VEL
LIN {X 0,Y 273.278,Z 567.758,A -85,B 0,C 180,E1 -18743.894,E2 -18743.894} C_VEL
LIN {X 0,Y 278.119,Z 558.521,A -85,B 0,C 180,E1 -18746.246,E2 -18746.246} C_VEL
LIN {X 0,Y 282.509,Z 549.151,A -85,B 0,C 180,E1 -18748.207,E2 -18748.207} C_VEL
LIN {X 0,Y 282.24,Z 544.324,A -85,B 0,C 180,E1 -18749.869,E2 -18749.869} C_VEL
LIN {X 0,Y 281.41,Z 539.503,A -85,B 0,C 180,E1 -18751.796,E2 -18751.796} C_VEL
LIN {X 0,Y 280.47,Z 537.575,A -85,B 0,C 180,E1 -18752.918,E2 -18752.918} C_VEL
LIN {X 0,Y 278.92,Z 536.583,A -85,B 0,C 180,E1 -18754.077,E2 -18754.077} C_VEL
LIN {X 0,Y 274.72,Z 535.707,A -85,B 0,C 180,E1 -18757.296,E2 -18757.296} C_VEL
LIN {X 0,Y 274.085,Z 535.267,A -85,B 0,C 180,E1 -18758.123,E2 -18758.123} C_VEL
LIN {X 0,Y 273.331,Z 534.073,A -85,B 0,C 180,E1 -18760.002,E2 -18760.002} C_VEL
LIN {X 0,Y 272.84,Z 533.424,A -85,B 0,C 180,E1 -18762.046,E2 -18762.046} C_VEL
LIN {X 0,Y 272.752,Z 533.361,A -85,B 0,C 180,E1 -18764.084,E2 -18764.084} C_VEL
LIN {X 0,Y 272.728,Z 534.559,A -85,B 0,C 180,E1 -18766.182,E2 -18766.182} C_VEL
LIN {X 0,Y 273.009,Z 538.071,A -85,B 0,C 180,E1 -18769.122,E2 -18769.122} C_VEL
LIN {X 0,Y 273.32,Z 540.164,A -85,B 0,C 180,E1 -18770.48,E2 -18770.48} C_VEL
LIN {X 0,Y 273.476,Z 544.606,A -85,B 0,C 180,E1 -18772.441,E2 -18772.441} C_VEL
LIN {X 0,Y 273.38,Z 550.478,A -85,B 0,C 180,E1 -18774.53,E2 -18774.53} C_VEL
LIN {X 0,Y 272.974,Z 557.938,A -85,B 0,C 180,E1 -18776.844,E2 -18776.844} C_VEL
LIN {X 0,Y 272.06,Z 565.359,A -85,B 0,C 180,E1 -18778.892,E2 -18778.892} C_VEL
LIN {X 0,Y 270.357,Z 572.831,A -85,B 0,C 180,E1 -18780.829,E2 -18780.829} C_VEL
LIN {X 0,Y 268.224,Z 578.795,A -85,B 0,C 180,E1 -18782.284,E2 -18782.284} C_VEL
LIN {X 0,Y 262.557,Z 589.686,A -85,B 0,C 180,E1 -18785.065,E2 -18785.065} C_VEL
LIN {X 0,Y 258.797,Z 596.456,A -85,B 0,C 180,E1 -18787.233,E2 -18787.233} C_VEL
LIN {X 0,Y 255.085,Z 603.02,A -85,B 0,C 180,E1 -18789.855,E2 -18789.855} C_VEL
LIN {X 0,Y 251.842,Z 608.924,A -85,B 0,C 180,E1 -18792.961,E2 -18792.961} C_VEL
LIN {X 0,Y 249.818,Z 612.354,A -85,B 0,C 180,E1 -18795.333,E2 -18795.333} C_VEL
LIN {X 0,Y 248.133,Z 615.623,A -85,B 0,C 180,E1 -18798.564,E2 -18798.564} C_VEL
LIN {X 0,Y 247.25,Z 617.424,A -85,B 0,C 180,E1 -18801.829,E2 -18801.829} C_VEL
LIN {X 0,Y 247.081,Z 617.735,A -85,B 0,C 180,E1 -18805.105,E2 -18805.105} C_VEL
LIN {X 0,Y 247.412,Z 616.549,A -85,B 0,C 180,E1 -18808.372,E2 -18808.372} C_VEL
LIN {X 0,Y 247.641,Z 615.32,A -85,B 0,C 180,E1 -18810,E2 -18810} C_VEL
LIN {X 0,Y 247.523,Z 612.605,A -85,B 0,C 180,E1 -18812.441,E2 -18812.441} C_VEL
LIN {X 0,Y 247.57,Z 608.83,A -85,B 0,C 180,E1 -18814.885,E2 -18814.885} C_VEL
LIN {X 0,Y 247.668,Z 604.048,A -85,B 0,C 180,E1 -18817.254,E2 -18817.254} C_VEL
LIN {X 0,Y 247.95,Z 597.503,A -85,B 0,C 180,E1 -18819.792,E2 -18819.792} C_VEL
LIN {X 0,Y 248.596,Z 589.657,A -85,B 0,C 180,E1 -18822.241,E2 -18822.241} C_VEL
LIN {X 0,Y 249.322,Z 581.707,A -85,B 0,C 180,E1 -18824.279,E2 -18824.279} C_VEL
LIN {X 0,Y 250.526,Z 571.107,A -85,B 0,C 180,E1 -18826.501,E2 -18826.501} C_VEL
LIN {X 0,Y 251.763,Z 560.194,A -85,B 0,C 180,E1 -18828.357,E2 -18828.357} C_VEL
LIN {X 0,Y 250.839,Z 549.492,A -85,B 0,C 180,E1 -18829.86,E2 -18829.86} C_VEL
LIN {X 0,Y 249.631,Z 536.644,A -85,B 0,C 180,E1 -18831.326,E2 -18831.326} C_VEL
LIN {X 0,Y 248.518,Z 522.974,A -85,B 0,C 180,E1 -18832.552,E2 -18832.552} C_VEL
LIN {X 0,Y 248.078,Z 514.666,A -85,B 0,C 180,E1 -18833.146,E2 -18833.146} C_VEL
LIN {X 0,Y 248.97,Z 508.684,A -85,B 0,C 180,E1 -18837.76,E2 -18837.76} C_VEL
LIN {X 0,Y 250.132,Z 502.504,A -85,B 0,C 180,E1 -18842.551,E2 -18842.551} C_VEL
LIN {X 0,Y 251.052,Z 498.085,A -85,B 0,C 180,E1 -18846.006,E2 -18846.006} C_VEL
LIN {X 0,Y 250.916,Z 495.197,A -85,B 0,C 180,E1 -18848.348,E2 -18848.348} C_VEL
LIN {X 0,Y 250.072,Z 490.383,A -85,B 0,C 180,E1 -18852.415,E2 -18852.415} C_VEL
LIN {X 0,Y 249.251,Z 485.439,A -85,B 0,C 180,E1 -18856.779,E2 -18856.779} C_VEL
LIN {X 0,Y 249.054,Z 485.458,A -85,B 0,C 180,E1 -18861.624,E2 -18861.624} C_VEL
LIN {X 0,Y 249.062,Z 485.458,A -85,B 0,C 180,E1 -18865.642,E2 -18865.642} C_VEL
LIN {X 0,Y 249.048,Z 485.459,A -85,B 0,C 180,E1 -18869.473,E2 -18869.473} C_VEL
LIN {X 0,Y 249.072,Z 485.458,A -85,B 0,C 180,E1 -18873.162,E2 -18873.162} C_VEL
LIN {X 0,Y 249.081,Z 485.459,A -85,B 0,C 180,E1 -18876.733,E2 -18876.733} C_VEL
LIN {X 0,Y 249.112,Z 485.452,A -85,B 0,C 180,E1 -18880.212,E2 -18880.212} C_VEL
LIN {X 0,Y 249.243,Z 485.436,A -85,B 0,C 180,E1 -18883.622,E2 -18883.622} C_VEL
LIN {X 0,Y 249.254,Z 485.436,A -85,B 0,C 180,E1 -18888.617,E2 -18888.617} C_VEL
LIN {X 0,Y 249.486,Z 485.406,A -85,B 0,C 180,E1 -18891.903,E2 -18891.903} C_VEL
LIN {X 0,Y 249.437,Z 485.412,A -85,B 0,C 180,E1 -18896.77,E2 -18896.77} C_VEL
LIN {X 0,Y 249.73,Z 485.375,A -85,B 0,C 180,E1 -18900,E2 -18900} C_VEL
LIN {X 0,Y 249.438,Z 485.412,A -85,B 0,C 180,E1 -18903.231,E2 -18903.231} C_VEL
LIN {X 0,Y 249.486,Z 485.406,A -85,B 0,C 180,E1 -18908.097,E2 -18908.097} C_VEL
LIN {X 0,Y 249.255,Z 485.434,A -85,B 0,C 180,E1 -18911.384,E2 -18911.384} C_VEL
LIN {X 0,Y 249.244,Z 485.437,A -85,B 0,C 180,E1 -18916.378,E2 -18916.378} C_VEL
LIN {X 0,Y 249.089,Z 485.455,A -85,B 0,C 180,E1 -18921.518,E2 -18921.518} C_VEL
LIN {X 0,Y 249.133,Z 485.448,A -85,B 0,C 180,E1 -18925.483,E2 -18925.483} C_VEL
LIN {X 0,Y 249.086,Z 485.456,A -85,B 0,C 180,E1 -18928.994,E2 -18928.994} C_VEL
LIN {X 0,Y 249.035,Z 485.463,A -85,B 0,C 180,E1 -18932.426,E2 -18932.426} C_VEL
LIN {X 0,Y 249.06,Z 485.463,A -85,B 0,C 180,E1 -18936.341,E2 -18936.341} C_VEL
LIN {X 0,Y 249.008,Z 485.466,A -85,B 0,C 180,E1 -18940.478,E2 -18940.478} C_VEL
LIN {X 0,Y 249.004,Z 485.466,A -85,B 0,C 180,E1 -18944.88,E2 -18944.88} C_VEL
LIN {X 0,Y 249.018,Z 485.464,A -85,B 0,C 180,E1 -18947.363,E2 -18947.363} C_VEL
LIN {X 0,Y 249.041,Z 485.46,A -85,B 0,C 180,E1 -18951.622,E2 -18951.622} C_VEL
LIN {X 0,Y 249.064,Z 485.459,A -85,B 0,C 180,E1 -18955.643,E2 -18955.643} C_VEL
LIN {X 0,Y 249.053,Z 485.457,A -85,B 0,C 180,E1 -18959.473,E2 -18959.473} C_VEL
LIN {X 0,Y 249.075,Z 485.457,A -85,B 0,C 180,E1 -18963.163,E2 -18963.163} C_VEL
LIN {X 0,Y 249.083,Z 485.455,A -85,B 0,C 180,E1 -18966.733,E2 -18966.733} C_VEL
LIN {X 0,Y 249.115,Z 485.455,A -85,B 0,C 180,E1 -18970.212,E2 -18970.212} C_VEL
LIN {X 0,Y 249.245,Z 485.437,A -85,B 0,C 180,E1 -18973.622,E2 -18973.622} C_VEL
LIN {X 0,Y 249.248,Z 485.435,A -85,B 0,C 180,E1 -18978.617,E2 -18978.617} C_VEL
LIN {X 0,Y 249.443,Z 485.414,A -85,B 0,C 180,E1 -18981.902,E2 -18981.902} C_VEL
LIN {X 0,Y 249.291,Z 485.428,A -85,B 0,C 180,E1 -18985.149,E2 -18985.149} C_VEL
LIN {X 0,Y 249.68,Z 485.383,A -85,B 0,C 180,E1 -18988.387,E2 -18988.387} C_VEL
LIN {X 0,Y 249.68,Z 485.383,A -85,B 0,C 180,E1 -18991.613,E2 -18991.613} C_VEL
LIN {X 0,Y 249.457,Z 485.41,A -85,B 0,C 180,E1 -18996.471,E2 -18996.471} C_VEL
LIN {X 0,Y 249.348,Z 485.426,A -85,B 0,C 180,E1 -18999.736,E2 -18999.736} C_VEL
LIN {X 0,Y 249.21,Z 485.439,A -85,B 0,C 180,E1 -19004.703,E2 -19004.703} C_VEL
LIN {X 0,Y 249.144,Z 485.451,A -85,B 0,C 180,E1 -19008.077,E2 -19008.077} C_VEL
LIN {X 0,Y 249.091,Z 485.455,A -85,B 0,C 180,E1 -19011.518,E2 -19011.518} C_VEL
LIN {X 0,Y 249.134,Z 485.451,A -85,B 0,C 180,E1 -19015.482,E2 -19015.482} C_VEL
LIN {X 0,Y 249.084,Z 485.455,A -85,B 0,C 180,E1 -19018.992,E2 -19018.992} C_VEL
LIN {X 0,Y 249.037,Z 485.461,A -85,B 0,C 180,E1 -19022.425,E2 -19022.425} C_VEL
LIN {X 0,Y 249.068,Z 485.458,A -85,B 0,C 180,E1 -19026.339,E2 -19026.339} C_VEL
LIN {X 0,Y 249.029,Z 485.461,A -85,B 0,C 180,E1 -19030.474,E2 -19030.474} C_VEL
LIN {X 0,Y 249.006,Z 485.465,A -85,B 0,C 180,E1 -19034.879,E2 -19034.879} C_VEL
LIN {X 0,Y 249.019,Z 485.464,A -85,B 0,C 180,E1 -19037.363,E2 -19037.363} C_VEL
LIN {X 0,Y 248.983,Z 485.471,A -85,B 0,C 180,E1 -19041.611,E2 -19041.611} C_VEL
LIN {X 0,Y 248.772,Z 485.498,A -85,B 0,C 180,E1 -19045.596,E2 -19045.596} C_VEL
LIN {X 0,Y 248.393,Z 485.543,A -85,B 0,C 180,E1 -19049.383,E2 -19049.383} C_VEL
LIN {X 0,Y 248.042,Z 485.589,A -85,B 0,C 180,E1 -19053.041,E2 -19053.041} C_VEL
LIN {X 0,Y 247.63,Z 485.684,A -85,B 0,C 180,E1 -19056.588,E2 -19056.588} C_VEL
LIN {X 0,Y 247.631,Z 486.132,A -85,B 0,C 180,E1 -19057.141,E2 -19057.141} C_VEL
LIN {X 0,Y 249.827,Z 499.098,A -85,B 0,C 180,E1 -19058.178,E2 -19058.178} C_VEL
LIN {X 0,Y 252.316,Z 513.021,A -85,B 0,C 180,E1 -19059.624,E2 -19059.624} C_VEL
LIN {X 0,Y 253.384,Z 518.965,A -85,B 0,C 180,E1 -19060.348,E2 -19060.348} C_VEL
LIN {X 0,Y 252.13,Z 532.05,A -85,B 0,C 180,E1 -19062.144,E2 -19062.144} C_VEL
LIN {X 0,Y 250.943,Z 542.695,A -85,B 0,C 180,E1 -19063.944,E2 -19063.944} C_VEL
LIN {X 0,Y 249.645,Z 553.328,A -85,B 0,C 180,E1 -19066.155,E2 -19066.155} C_VEL
LIN {X 0,Y 248.671,Z 562.878,A -85,B 0,C 180,E1 -19068.589,E2 -19068.589} C_VEL
LIN {X 0,Y 247.958,Z 570.586,A -85,B 0,C 180,E1 -19071.031,E2 -19071.031} C_VEL
LIN {X 0,Y 247.474,Z 577.421,A -85,B 0,C 180,E1 -19073.704,E2 -19073.704} C_VEL
LIN {X 0,Y 247.308,Z 582.002,A -85,B 0,C 180,E1 -19075.926,E2 -19075.926} C_VEL
LIN {X 0,Y 247.193,Z 586.018,A -85,B 0,C 180,E1 -19078.371,E2 -19078.371} C_VEL
LIN {X 0,Y 247.197,Z 588.146,A -85,B 0,C 180,E1 -19080,E2 -19080} C_VEL
LIN {X 0,Y 247.338,Z 589.851,A -85,B 0,C 180,E1 -19081.628,E2 -19081.628} C_VEL
LIN {X 0,Y 247.95,Z 592.041,A -85,B 0,C 180,E1 -19084.878,E2 -19084.878} C_VEL
LIN {X 0,Y 248.888,Z 592.766,A -85,B 0,C 180,E1 -19088.116,E2 -19088.116} C_VEL
LIN {X 0,Y 250.753,Z 591.956,A -85,B 0,C 180,E1 -19091.314,E2 -19091.314} C_VEL
LIN {X 0,Y 253.11,Z 589.701,A -85,B 0,C 180,E1 -19094.471,E2 -19094.471} C_VEL
LIN {X 0,Y 255.508,Z 587.027,A -85,B 0,C 180,E1 -19096.787,E2 -19096.787} C_VEL
LIN {X 0,Y 258.23,Z 583.474,A -85,B 0,C 180,E1 -19099.062,E2 -19099.062} C_VEL
LIN {X 0,Y 262.575,Z 577.305,A -85,B 0,C 180,E1 -19102.007,E2 -19102.007} C_VEL
LIN {X 0,Y 267.116,Z 570.265,A -85,B 0,C 180,E1 -19104.481,E2 -19104.481} C_VEL
LIN {X 0,Y 272.21,Z 561.68,A -85,B 0,C 180,E1 -19106.86,E2 -19106.86} C_VEL
LIN {X 0,Y 276.877,Z 552.703,A -85,B 0,C 180,E1 -19108.834,E2 -19108.834} C_VEL
LIN {X 0,Y 277.115,Z 550.079,A -85,B 0,C 180,E1 -19109.761,E2 -19109.761} C_VEL
LIN {X 0,Y 276.556,Z 544.201,A -85,B 0,C 180,E1 -19112.253,E2 -19112.253} C_VEL
LIN {X 0,Y 275.866,Z 540.584,A -85,B 0,C 180,E1 -19114.089,E2 -19114.089} C_VEL
LIN {X 0,Y 275.048,Z 537.551,A -85,B 0,C 180,E1 -19115.993,E2 -19115.993} C_VEL
LIN {X 0,Y 274.085,Z 535.267,A -85,B 0,C 180,E1 -19118.123,E2 -19118.123} C_VEL
LIN {X 0,Y 273.231,Z 535.085,A -85,B 0,C 180,E1 -19119.344,E2 -19119.344} C_VEL
LIN {X 0,Y 271.989,Z 535.891,A -85,B 0,C 180,E1 -19120.553,E2 -19120.553} C_VEL
LIN {X 0,Y 269.533,Z 538.608,A -85,B 0,C 180,E1 -19122.977,E2 -19122.977} C_VEL
LIN {X 0,Y 268.908,Z 539.598,A -85,B 0,C 180,E1 -19124.23,E2 -19124.23} C_VEL
LIN {X 0,Y 268.868,Z 539.756,A -85,B 0,C 180,E1 -19124.655,E2 -19124.655} C_VEL
LIN {X 0,Y 268.833,Z 541.703,A -85,B 0,C 180,E1 -19127.179,E2 -19127.179} C_VEL
LIN {X 0,Y 268.993,Z 544.291,A -85,B 0,C 180,E1 -19129.261,E2 -19129.261} C_VEL
LIN {X 0,Y 269.076,Z 546.178,A -85,B 0,C 180,E1 -19130.399,E2 -19130.399} C_VEL
LIN {X 0,Y 268.86,Z 551.012,A -85,B 0,C 180,E1 -19132.541,E2 -19132.541} C_VEL
LIN {X 0,Y 268.103,Z 558.878,A -85,B 0,C 180,E1 -19135.322,E2 -19135.322} C_VEL
LIN {X 0,Y 266.924,Z 566.451,A -85,B 0,C 180,E1 -19137.655,E2 -19137.655} C_VEL
LIN {X 0,Y 265.052,Z 573.93,A -85,B 0,C 180,E1 -19139.748,E2 -19139.748} C_VEL
LIN {X 0,Y 263.535,Z 578.096,A -85,B 0,C 180,E1 -19140.876,E2 -19140.876} C_VEL
LIN {X 0,Y 259.177,Z 586.321,A -85,B 0,C 180,E1 -19142.986,E2 -19142.986} C_VEL
LIN {X 0,Y 253.545,Z 595.588,A -85,B 0,C 180,E1 -19145.867,E2 -19145.867} C_VEL
LIN {X 0,Y 249.437,Z 602.156,A -85,B 0,C 180,E1 -19148.513,E2 -19148.513} C_VEL
LIN {X 0,Y 245.833,Z 608.076,A -85,B 0,C 180,E1 -19151.671,E2 -19151.671} C_VEL
LIN {X 0,Y 242.966,Z 612.517,A -85,B 0,C 180,E1 -19154.91,E2 -19154.91} C_VEL
LIN {X 0,Y 241.157,Z 615.47,A -85,B 0,C 180,E1 -19158.229,E2 -19158.229} C_VEL
LIN {X 0,Y 240.199,Z 617.007,A -85,B 0,C 180,E1 -19161.587,E2 -19161.587} C_VEL
LIN {X 0,Y 240.011,Z 617.109,A -85,B 0,C 180,E1 -19164.96,E2 -19164.96} C_VEL
LIN {X 0,Y 240.365,Z 615.661,A -85,B 0,C 180,E1 -19168.324,E2 -19168.324} C_VEL
LIN {X 0,Y 240.626,Z 614.342,A -85,B 0,C 180,E1 -19170,E2 -19170} C_VEL
LIN {X 0,Y 240.505,Z 611.425,A -85,B 0,C 180,E1 -19172.512,E2 -19172.512} C_VEL
LIN {X 0,Y 240.552,Z 607.435,A -85,B 0,C 180,E1 -19175.028,E2 -19175.028} C_VEL
LIN {X 0,Y 240.673,Z 602.439,A -85,B 0,C 180,E1 -19177.466,E2 -19177.466} C_VEL
LIN {X 0,Y 240.971,Z 595.71,A -85,B 0,C 180,E1 -19180.078,E2 -19180.078} C_VEL
LIN {X 0,Y 241.667,Z 587.637,A -85,B 0,C 180,E1 -19182.598,E2 -19182.598} C_VEL
LIN {X 0,Y 242.625,Z 577.523,A -85,B 0,C 180,E1 -19185.111,E2 -19185.111} C_VEL
LIN {X 0,Y 243.832,Z 567.223,A -85,B 0,C 180,E1 -19187.184,E2 -19187.184} C_VEL
LIN {X 0,Y 244.619,Z 559.174,A -85,B 0,C 180,E1 -19188.54,E2 -19188.54} C_VEL
LIN {X 0,Y 243.458,Z 546.913,A -85,B 0,C 180,E1 -19190.268,E2 -19190.268} C_VEL
LIN {X 0,Y 242.228,Z 533.397,A -85,B 0,C 180,E1 -19191.806,E2 -19191.806} C_VEL
LIN {X 0,Y 241.226,Z 519.39,A -85,B 0,C 180,E1 -19193.019,E2 -19193.019} C_VEL
LIN {X 0,Y 241.009,Z 514.297,A -85,B 0,C 180,E1 -19193.41,E2 -19193.41} C_VEL
LIN {X 0,Y 242.065,Z 507.806,A -85,B 0,C 180,E1 -19198.597,E2 -19198.597} C_VEL
LIN {X 0,Y 243.238,Z 501.953,A -85,B 0,C 180,E1 -19203.297,E2 -19203.297} C_VEL
LIN {X 0,Y 243.978,Z 498.32,A -85,B 0,C 180,E1 -19206.238,E2 -19206.238} C_VEL
LIN {X 0,Y 243.671,Z 494.571,A -85,B 0,C 180,E1 -19209.385,E2 -19209.385} C_VEL
LIN {X 0,Y 242.74,Z 489.751,A -85,B 0,C 180,E1 -19213.629,E2 -19213.629} C_VEL
LIN {X 0,Y 242.2,Z 486.316,A -85,B 0,C 180,E1 -19216.898,E2 -19216.898} C_VEL
LIN {X 0,Y 242.013,Z 486.337,A -85,B 0,C 180,E1 -19222.423,E2 -19222.423} C_VEL
LIN {X 0,Y 241.992,Z 486.342,A -85,B 0,C 180,E1 -19226.509,E2 -19226.509} C_VEL
LIN {X 0,Y 242.014,Z 486.338,A -85,B 0,C 180,E1 -19230.597,E2 -19230.597} C_VEL
LIN {X 0,Y 242.068,Z 486.33,A -85,B 0,C 180,E1 -19234.183,E2 -19234.183} C_VEL
LIN {X 0,Y 242.054,Z 486.333,A -85,B 0,C 180,E1 -19238.297,E2 -19238.297} C_VEL
LIN {X 0,Y 242.164,Z 486.318,A -85,B 0,C 180,E1 -19243.278,E2 -19243.278} C_VEL
LIN {X 0,Y 242.188,Z 486.316,A -85,B 0,C 180,E1 -19248.28,E2 -19248.28} C_VEL
LIN {X 0,Y 242.437,Z 486.283,A -85,B 0,C 180,E1 -19251.666,E2 -19251.666} C_VEL
LIN {X 0,Y 242.261,Z 486.306,A -85,B 0,C 180,E1 -19255.007,E2 -19255.007} C_VEL
LIN {X 0,Y 242.638,Z 486.259,A -85,B 0,C 180,E1 -19258.34,E2 -19258.34} C_VEL
LIN {X 0,Y 242.639,Z 486.259,A -85,B 0,C 180,E1 -19261.66,E2 -19261.66} C_VEL
LIN {X 0,Y 242.431,Z 486.285,A -85,B 0,C 180,E1 -19266.734,E2 -19266.734} C_VEL
LIN {X 0,Y 242.347,Z 486.296,A -85,B 0,C 180,E1 -19270.021,E2 -19270.021} C_VEL
LIN {X 0,Y 242.169,Z 486.314,A -85,B 0,C 180,E1 -19275.141,E2 -19275.141} C_VEL
LIN {X 0,Y 242.075,Z 486.332,A -85,B 0,C 180,E1 -19278.624,E2 -19278.624} C_VEL
LIN {X 0,Y 242.015,Z 486.339,A -85,B 0,C 180,E1 -19282.18,E2 -19282.18} C_VEL
LIN {X 0,Y 242.068,Z 486.329,A -85,B 0,C 180,E1 -19285.838,E2 -19285.838} C_VEL
LIN {X 0,Y 242.032,Z 486.334,A -85,B 0,C 180,E1 -19289.58,E2 -19289.58} C_VEL
LIN {X 0,Y 241.99,Z 486.337,A -85,B 0,C 180,E1 -19293.492,E2 -19293.492} C_VEL
LIN {X 0,Y 241.993,Z 486.339,A -85,B 0,C 180,E1 -19297.582,E2 -19297.582} C_VEL
LIN {X 0,Y 241.939,Z 486.345,A -85,B 0,C 180,E1 -19301.923,E2 -19301.923} C_VEL
LIN {X 0,Y 241.936,Z 486.348,A -85,B 0,C 180,E1 -19306.572,E2 -19306.572} C_VEL
LIN {X 0,Y 241.975,Z 486.342,A -85,B 0,C 180,E1 -19310.285,E2 -19310.285} C_VEL
LIN {X 0,Y 242.039,Z 486.336,A -85,B 0,C 180,E1 -19314.498,E2 -19314.498} C_VEL
LIN {X 0,Y 241.979,Z 486.34,A -85,B 0,C 180,E1 -19318.481,E2 -19318.481} C_VEL
LIN {X 0,Y 242.01,Z 486.34,A -85,B 0,C 180,E1 -19322.313,E2 -19322.313} C_VEL
LIN {X 0,Y 242.061,Z 486.334,A -85,B 0,C 180,E1 -19326.016,E2 -19326.016} C_VEL
LIN {X 0,Y 242.041,Z 486.332,A -85,B 0,C 180,E1 -19329.608,E2 -19329.608} C_VEL
LIN {X 0,Y 242.167,Z 486.318,A -85,B 0,C 180,E1 -19333.279,E2 -19333.279} C_VEL
LIN {X 0,Y 242.185,Z 486.317,A -85,B 0,C 180,E1 -19338.28,E2 -19338.28} C_VEL
LIN {X 0,Y 242.392,Z 486.291,A -85,B 0,C 180,E1 -19341.665,E2 -19341.665} C_VEL
LIN {X 0,Y 242.252,Z 486.304,A -85,B 0,C 180,E1 -19345.007,E2 -19345.007} C_VEL
LIN {X 0,Y 242.64,Z 486.26,A -85,B 0,C 180,E1 -19348.34,E2 -19348.34} C_VEL
LIN {X 0,Y 242.64,Z 486.26,A -85,B 0,C 180,E1 -19351.66,E2 -19351.66} C_VEL
LIN {X 0,Y 242.428,Z 486.285,A -85,B 0,C 180,E1 -19356.659,E2 -19356.659} C_VEL
LIN {X 0,Y 242.272,Z 486.307,A -85,B 0,C 180,E1 -19360.024,E2 -19360.024} C_VEL
LIN {X 0,Y 242.171,Z 486.316,A -85,B 0,C 180,E1 -19365.141,E2 -19365.141} C_VEL
LIN {X 0,Y 242.078,Z 486.329,A -85,B 0,C 180,E1 -19368.624,E2 -19368.624} C_VEL
LIN {X 0,Y 242.017,Z 486.336,A -85,B 0,C 180,E1 -19372.18,E2 -19372.18} C_VEL
LIN {X 0,Y 242.07,Z 486.333,A -85,B 0,C 180,E1 -19375.838,E2 -19375.838} C_VEL
LIN {X 0,Y 242.033,Z 486.336,A -85,B 0,C 180,E1 -19379.58,E2 -19379.58} C_VEL
LIN {X 0,Y 241.992,Z 486.34,A -85,B 0,C 180,E1 -19383.491,E2 -19383.491} C_VEL
LIN {X 0,Y 242.002,Z 486.34,A -85,B 0,C 180,E1 -19387.58,E2 -19387.58} C_VEL
LIN {X 0,Y 241.946,Z 486.348,A -85,B 0,C 180,E1 -19391.921,E2 -19391.921} C_VEL
LIN {X 0,Y 241.937,Z 486.345,A -85,B 0,C 180,E1 -19396.571,E2 -19396.571} C_VEL
LIN {X 0,Y 241.936,Z 486.346,A -85,B 0,C 180,E1 -19400.276,E2 -19400.276} C_VEL
LIN {X 0,Y 241.909,Z 486.35,A -85,B 0,C 180,E1 -19402.403,E2 -19402.403} C_VEL
LIN {X 0,Y 241.616,Z 486.384,A -85,B 0,C 180,E1 -19406.45,E2 -19406.45} C_VEL
LIN {X 0,Y 241.228,Z 486.435,A -85,B 0,C 180,E1 -19410.931,E2 -19410.931} C_VEL
LIN {X 0,Y 240.681,Z 486.509,A -85,B 0,C 180,E1 -19415.87,E2 -19415.87} C_VEL
LIN {X 0,Y 240.568,Z 486.521,A -85,B 0,C 180,E1 -19416.885,E2 -19416.885} C_VEL
LIN {X 0,Y 242.817,Z 500.04,A -85,B 0,C 180,E1 -19418.015,E2 -19418.015} C_VEL
LIN {X 0,Y 245.227,Z 513.525,A -85,B 0,C 180,E1 -19419.469,E2 -19419.469} C_VEL
LIN {X 0,Y 246.258,Z 519.3,A -85,B 0,C 180,E1 -19420.195,E2 -19420.195} C_VEL
LIN {X 0,Y 245.033,Z 532.374,A -85,B 0,C 180,E1 -19422.041,E2 -19422.041} C_VEL
LIN {X 0,Y 243.84,Z 542.976,A -85,B 0,C 180,E1 -19423.894,E2 -19423.894} C_VEL
LIN {X 0,Y 242.533,Z 553.553,A -85,B 0,C 180,E1 -19426.168,E2 -19426.168} C_VEL
LIN {X 0,Y 241.562,Z 563.093,A -85,B 0,C 180,E1 -19428.674,E2 -19428.674} C_VEL
LIN {X 0,Y 240.853,Z 570.859,A -85,B 0,C 180,E1 -19431.188,E2 -19431.188} C_VEL
LIN {X 0,Y 240.387,Z 577.294,A -85,B 0,C 180,E1 -19433.741,E2 -19433.741} C_VEL
LIN {X 0,Y 240.182,Z 583.102,A -85,B 0,C 180,E1 -19436.645,E2 -19436.645} C_VEL
LIN {X 0,Y 240.095,Z 586.95,A -85,B 0,C 180,E1 -19439.161,E2 -19439.161} C_VEL
LIN {X 0,Y 240.263,Z 589.846,A -85,B 0,C 180,E1 -19441.676,E2 -19441.676} C_VEL
LIN {X 0,Y 240.53,Z 591.292,A -85,B 0,C 180,E1 -19443.35,E2 -19443.35} C_VEL
LIN {X 0,Y 240.899,Z 592.342,A -85,B 0,C 180,E1 -19445.021,E2 -19445.021} C_VEL
LIN {X 0,Y 241.889,Z 593.299,A -85,B 0,C 180,E1 -19448.353,E2 -19448.353} C_VEL
LIN {X 0,Y 243.864,Z 592.794,A -85,B 0,C 180,E1 -19451.638,E2 -19451.638} C_VEL
LIN {X 0,Y 246.341,Z 590.858,A -85,B 0,C 180,E1 -19454.878,E2 -19454.878} C_VEL
LIN {X 0,Y 249.727,Z 587.42,A -85,B 0,C 180,E1 -19458.033,E2 -19458.033} C_VEL
LIN {X 0,Y 252.845,Z 583.846,A -85,B 0,C 180,E1 -19460.331,E2 -19460.331} C_VEL
LIN {X 0,Y 256.269,Z 579.357,A -85,B 0,C 180,E1 -19462.578,E2 -19462.578} C_VEL
LIN {X 0,Y 261.006,Z 572.844,A -85,B 0,C 180,E1 -19465.093,E2 -19465.093} C_VEL
LIN {X 0,Y 266.307,Z 564.684,A -85,B 0,C 180,E1 -19467.505,E2 -19467.505} C_VEL
LIN {X 0,Y 271.201,Z 556.389,A -85,B 0,C 180,E1 -19469.497,E2 -19469.497} C_VEL
LIN {X 0,Y 271.735,Z 554.948,A -85,B 0,C 180,E1 -19469.918,E2 -19469.918} C_VEL
LIN {X 0,Y 271.624,Z 549.339,A -85,B 0,C 180,E1 -19472.445,E2 -19472.445} C_VEL
LIN {X 0,Y 271.115,Z 545.172,A -85,B 0,C 180,E1 -19474.771,E2 -19474.771} C_VEL
LIN {X 0,Y 270.518,Z 542.548,A -85,B 0,C 180,E1 -19476.693,E2 -19476.693} C_VEL
LIN {X 0,Y 269.823,Z 540.743,A -85,B 0,C 180,E1 -19478.691,E2 -19478.691} C_VEL
LIN {X 0,Y 269.194,Z 539.737,A -85,B 0,C 180,E1 -19480.789,E2 -19480.789} C_VEL
LIN {X 0,Y 268.945,Z 539.352,A -85,B 0,C 180,E1 -19482.971,E2 -19482.971} C_VEL
LIN {X 0,Y 268.868,Z 539.756,A -85,B 0,C 180,E1 -19484.655,E2 -19484.655} C_VEL
LIN {X 0,Y 268.769,Z 540.329,A -85,B 0,C 180,E1 -19485.482,E2 -19485.482} C_VEL
LIN {X 0,Y 268.063,Z 542.266,A -85,B 0,C 180,E1 -19486.665,E2 -19486.665} C_VEL
LIN {X 0,Y 267.017,Z 544.995,A -85,B 0,C 180,E1 -19487.779,E2 -19487.779} C_VEL
LIN {X 0,Y 264.819,Z 551.201,A -85,B 0,C 180,E1 -19490.011,E2 -19490.011} C_VEL
LIN {X 0,Y 264.44,Z 552.98,A -85,B 0,C 180,E1 -19490.801,E2 -19490.801} C_VEL
LIN {X 0,Y 263.683,Z 558.425,A -85,B 0,C 180,E1 -19493.091,E2 -19493.091} C_VEL
LIN {X 0,Y 262.691,Z 564.171,A -85,B 0,C 180,E1 -19495.162,E2 -19495.162} C_VEL
LIN {X 0,Y 261.055,Z 571.154,A -85,B 0,C 180,E1 -19497.423,E2 -19497.423} C_VEL
LIN {X 0,Y 258.847,Z 577.738,A -85,B 0,C 180,E1 -19499.397,E2 -19499.397} C_VEL
LIN {X 0,Y 256.212,Z 583.032,A -85,B 0,C 180,E1 -19500.863,E2 -19500.863} C_VEL
LIN {X 0,Y 250.013,Z 592.696,A -85,B 0,C 180,E1 -19503.721,E2 -19503.721} C_VEL
LIN {X 0,Y 245.301,Z 599.587,A -85,B 0,C 180,E1 -19506.352,E2 -19506.352} C_VEL
LIN {X 0,Y 241.896,Z 604.51,A -85,B 0,C 180,E1 -19508.705,E2 -19508.705} C_VEL
LIN {X 0,Y 238.319,Z 609.67,A -85,B 0,C 180,E1 -19511.962,E2 -19511.962} C_VEL
LIN {X 0,Y 236.099,Z 612.61,A -85,B 0,C 180,E1 -19514.46,E2 -19514.46} C_VEL
LIN {X 0,Y 234.176,Z 615.286,A -85,B 0,C 180,E1 -19517.873,E2 -19517.873} C_VEL
LIN {X 0,Y 233.169,Z 616.576,A -85,B 0,C 180,E1 -19521.332,E2 -19521.332} C_VEL
LIN {X 0,Y 232.969,Z 616.396,A -85,B 0,C 180,E1 -19524.807,E2 -19524.807} C_VEL
LIN {X 0,Y 233.317,Z 614.725,A -85,B 0,C 180,E1 -19528.274,E2 -19528.274} C_VEL
LIN {X 0,Y 233.608,Z 613.308,A -85,B 0,C 180,E1 -19530,E2 -19530} C_VEL
LIN {X 0,Y 233.505,Z 610.226,A -85,B 0,C 180,E1 -19532.587,E2 -19532.587} C_VEL
LIN {X 0,Y 233.538,Z 606.042,A -85,B 0,C 180,E1 -19535.18,E2 -19535.18} C_VEL
LIN {X 0,Y 233.745,Z 599.56,A -85,B 0,C 180,E1 -19538.211,E2 -19538.211} C_VEL
LIN {X 0,Y 234.096,Z 592.474,A -85,B 0,C 180,E1 -19540.815,E2 -19540.815} C_VEL
LIN {X 0,Y 234.888,Z 583.777,A -85,B 0,C 180,E1 -19543.408,E2 -19543.408} C_VEL
LIN {X 0,Y 236.031,Z 572.947,A -85,B 0,C 180,E1 -19545.987,E2 -19545.987} C_VEL
LIN {X 0,Y 237.301,Z 562.1,A -85,B 0,C 180,E1 -19548.068,E2 -19548.068} C_VEL
LIN {X 0,Y 237.433,Z 558.311,A -85,B 0,C 180,E1 -19548.702,E2 -19548.702} C_VEL
LIN {X 0,Y 236.245,Z 546.143,A -85,B 0,C 180,E1 -19550.46,E2 -19550.46} C_VEL
LIN {X 0,Y 235.066,Z 532.428,A -85,B 0,C 180,E1 -19552.053,E2 -19552.053} C_VEL
LIN {X 0,Y 234.156,Z 519.661,A -85,B 0,C 180,E1 -19553.2,E2 -19553.2} C_VEL
LIN {X 0,Y 233.958,Z 513.94,A -85,B 0,C 180,E1 -19553.631,E2 -19553.631} C_VEL
LIN {X 0,Y 234.967,Z 507.96,A -85,B 0,C 180,E1 -19558.592,E2 -19558.592} C_VEL
LIN {X 0,Y 236.199,Z 501.966,A -85,B 0,C 180,E1 -19563.579,E2 -19563.579} C_VEL
LIN {X 0,Y 236.908,Z 498.606,A -85,B 0,C 180,E1 -19566.392,E2 -19566.392} C_VEL
LIN {X 0,Y 236.583,Z 495.12,A -85,B 0,C 180,E1 -19569.434,E2 -19569.434} C_VEL
LIN {X 0,Y 235.778,Z 490.865,A -85,B 0,C 180,E1 -19573.281,E2 -19573.281} C_VEL
LIN {X 0,Y 235.178,Z 487.192,A -85,B 0,C 180,E1 -19576.832,E2 -19576.832} C_VEL
LIN {X 0,Y 234.971,Z 487.214,A -85,B 0,C 180,E1 -19581.089,E2 -19581.089} C_VEL
LIN {X 0,Y 234.961,Z 487.215,A -85,B 0,C 180,E1 -19585.367,E2 -19585.367} C_VEL
LIN {X 0,Y 234.923,Z 487.219,A -85,B 0,C 180,E1 -19589.431,E2 -19589.431} C_VEL
LIN {X 0,Y 234.994,Z 487.21,A -85,B 0,C 180,E1 -19593.794,E2 -19593.794} C_VEL
LIN {X 0,Y 235.012,Z 487.208,A -85,B 0,C 180,E1 -19598.97,E2 -19598.97} C_VEL
LIN {X 0,Y 235.097,Z 487.199,A -85,B 0,C 180,E1 -19603.059,E2 -19603.059} C_VEL
LIN {X 0,Y 235.148,Z 487.191,A -85,B 0,C 180,E1 -19607.924,E2 -19607.924} C_VEL
LIN {X 0,Y 235.392,Z 487.161,A -85,B 0,C 180,E1 -19611.415,E2 -19611.415} C_VEL
LIN {X 0,Y 235.407,Z 487.16,A -85,B 0,C 180,E1 -19613.142,E2 -19613.142} C_VEL
LIN {X 0,Y 235.598,Z 487.135,A -85,B 0,C 180,E1 -19618.291,E2 -19618.291} C_VEL
LIN {X 0,Y 235.598,Z 487.136,A -85,B 0,C 180,E1 -19621.71,E2 -19621.71} C_VEL
LIN {X 0,Y 235.408,Z 487.159,A -85,B 0,C 180,E1 -19626.859,E2 -19626.859} C_VEL
LIN {X 0,Y 235.255,Z 487.181,A -85,B 0,C 180,E1 -19630.326,E2 -19630.326} C_VEL
LIN {X 0,Y 235.116,Z 487.193,A -85,B 0,C 180,E1 -19635.607,E2 -19635.607} C_VEL
LIN {X 0,Y 235.011,Z 487.209,A -85,B 0,C 180,E1 -19639.206,E2 -19639.206} C_VEL
LIN {X 0,Y 234.963,Z 487.214,A -85,B 0,C 180,E1 -19642.883,E2 -19642.883} C_VEL
LIN {X 0,Y 234.972,Z 487.216,A -85,B 0,C 180,E1 -19646.658,E2 -19646.658} C_VEL
LIN {X 0,Y 234.934,Z 487.22,A -85,B 0,C 180,E1 -19650.568,E2 -19650.568} C_VEL
LIN {X 0,Y 234.944,Z 487.219,A -85,B 0,C 180,E1 -19654.636,E2 -19654.636} C_VEL
LIN {X 0,Y 234.943,Z 487.217,A -85,B 0,C 180,E1 -19658.945,E2 -19658.945} C_VEL
LIN {X 0,Y 234.889,Z 487.223,A -85,B 0,C 180,E1 -19663.486,E2 -19663.486} C_VEL
LIN {X 0,Y 234.889,Z 487.226,A -85,B 0,C 180,E1 -19666.515,E2 -19666.515} C_VEL
LIN {X 0,Y 234.957,Z 487.213,A -85,B 0,C 180,E1 -19671.086,E2 -19671.086} C_VEL
LIN {X 0,Y 234.963,Z 487.215,A -85,B 0,C 180,E1 -19675.368,E2 -19675.368} C_VEL
LIN {X 0,Y 234.971,Z 487.215,A -85,B 0,C 180,E1 -19680.158,E2 -19680.158} C_VEL
LIN {X 0,Y 234.997,Z 487.212,A -85,B 0,C 180,E1 -19683.794,E2 -19683.794} C_VEL
LIN {X 0,Y 235.015,Z 487.206,A -85,B 0,C 180,E1 -19688.97,E2 -19688.97} C_VEL
LIN {X 0,Y 235.1,Z 487.198,A -85,B 0,C 180,E1 -19693.06,E2 -19693.06} C_VEL
LIN {X 0,Y 235.119,Z 487.196,A -85,B 0,C 180,E1 -19697.922,E2 -19697.922} C_VEL
LIN {X 0,Y 235.325,Z 487.17,A -85,B 0,C 180,E1 -19701.412,E2 -19701.412} C_VEL
LIN {X 0,Y 235.364,Z 487.164,A -85,B 0,C 180,E1 -19703.14,E2 -19703.14} C_VEL
LIN {X 0,Y 235.599,Z 487.138,A -85,B 0,C 180,E1 -19708.291,E2 -19708.291} C_VEL
LIN {X 0,Y 235.6,Z 487.138,A -85,B 0,C 180,E1 -19711.71,E2 -19711.71} C_VEL
LIN {X 0,Y 235.378,Z 487.163,A -85,B 0,C 180,E1 -19716.86,E2 -19716.86} C_VEL
LIN {X 0,Y 235.218,Z 487.184,A -85,B 0,C 180,E1 -19720.328,E2 -19720.328} C_VEL
LIN {X 0,Y 235.118,Z 487.196,A -85,B 0,C 180,E1 -19725.606,E2 -19725.606} C_VEL
LIN {X 0,Y 235.013,Z 487.209,A -85,B 0,C 180,E1 -19729.205,E2 -19729.205} C_VEL
LIN {X 0,Y 234.965,Z 487.212,A -85,B 0,C 180,E1 -19732.883,E2 -19732.883} C_VEL
LIN {X 0,Y 234.973,Z 487.214,A -85,B 0,C 180,E1 -19736.657,E2 -19736.657} C_VEL
LIN {X 0,Y 234.935,Z 487.215,A -85,B 0,C 180,E1 -19740.568,E2 -19740.568} C_VEL
LIN {X 0,Y 234.963,Z 487.215,A -85,B 0,C 180,E1 -19744.633,E2 -19744.633} C_VEL
LIN {X 0,Y 234.945,Z 487.215,A -85,B 0,C 180,E1 -19748.944,E2 -19748.944} C_VEL
LIN {X 0,Y 234.89,Z 487.226,A -85,B 0,C 180,E1 -19753.486,E2 -19753.486} C_VEL
LIN {X 0,Y 234.89,Z 487.223,A -85,B 0,C 180,E1 -19756.514,E2 -19756.514} C_VEL
LIN {X 0,Y 234.889,Z 487.224,A -85,B 0,C 180,E1 -19761.072,E2 -19761.072} C_VEL
LIN {X 0,Y 234.64,Z 487.256,A -85,B 0,C 180,E1 -19765.312,E2 -19765.312} C_VEL
LIN {X 0,Y 234.275,Z 487.301,A -85,B 0,C 180,E1 -19769.337,E2 -19769.337} C_VEL
LIN {X 0,Y 233.878,Z 487.353,A -85,B 0,C 180,E1 -19773.208,E2 -19773.208} C_VEL
LIN {X 0,Y 233.521,Z 487.399,A -85,B 0,C 180,E1 -19776.704,E2 -19776.704} C_VEL
LIN {X 0,Y 235.96,Z 501.894,A -85,B 0,C 180,E1 -19777.98,E2 -19777.98} C_VEL
LIN {X 0,Y 238.239,Z 514.74,A -85,B 0,C 180,E1 -19779.423,E2 -19779.423} C_VEL
LIN {X 0,Y 239.165,Z 520.001,A -85,B 0,C 180,E1 -19780.109,E2 -19780.109} C_VEL
LIN {X 0,Y 237.949,Z 532.428,A -85,B 0,C 180,E1 -19781.933,E2 -19781.933} C_VEL
LIN {X 0,Y 236.738,Z 543.051,A -85,B 0,C 180,E1 -19783.84,E2 -19783.84} C_VEL
LIN {X 0,Y 235.403,Z 553.703,A -85,B 0,C 180,E1 -19786.181,E2 -19786.181} C_VEL
LIN {X 0,Y 234.437,Z 563.299,A -85,B 0,C 180,E1 -19788.763,E2 -19788.763} C_VEL
LIN {X 0,Y 233.732,Z 571.12,A -85,B 0,C 180,E1 -19791.353,E2 -19791.353} C_VEL
LIN {X 0,Y 233.214,Z 578.267,A -85,B 0,C 180,E1 -19794.318,E2 -19794.318} C_VEL
